	{attribute 'TcIecLibraryType'}
	{attribute 'external_name' := 'F_VN_AppendToContainer_ITcVnForwardIterator_GUID_EB72DC2C_3543_2E88_7126_C09EBB4E7DA0'}
	(* Append a single element (represented by an iterator)to a container. *)
	FUNCTION F_VN_AppendToContainer_ITcVnForwardIterator : HRESULT
	VAR_INPUT
		ipElement	:	ITcVnForwardIterator;	(* Single element to append to ipContainer *)
		ipContainer	:	ITcVnContainer;	(* Container to which the element(s) will be appended *)
		hrPrev	:	HRESULT;	(* HRESULT indicating the result of previous operations (If SUCCEEDED(hrPrev) equals false, no operation is executed.) *)
	END_VAR

END_FUNCTION

// Functions/Basic Container Operations/F_VN_AppendToContainer/F_VN_AppendToContainer_DINT

	{attribute 'TcIecLibraryType'}
	{attribute 'external_name' := 'F_VN_AppendToContainer_DINT_GUID_466F0C35_D3B5_2E85_68F4_3D84EB5E34A6'}
	(* Append a single element of type DINT to a container. *)
	FUNCTION F_VN_AppendToContainer_DINT : HRESULT
	VAR_INPUT
		nElement	:	DINT;	(* Single element to append to ipContainer *)
		ipContainer	:	ITcVnContainer;	(* Container to which the element will be appended *)
		hrPrev	:	HRESULT;	(* HRESULT indicating the result of previous operations (If SUCCEEDED(hrPrev) equals false, no operation is executed.) *)
	END_VAR

END_FUNCTION

// Functions/Basic Container Operations/F_VN_AppendToContainer/F_VN_AppendToContainer_INT

	{attribute 'TcIecLibraryType'}
	{attribute 'external_name' := 'F_VN_AppendToContainer_INT_GUID_9C2E93C7_B738_2FE7_7542_11A5629F66B3'}
	(* Append a single element of type INT to a container. *)
	FUNCTION F_VN_AppendToContainer_INT : HRESULT
	VAR_INPUT
		nElement	:	INT;	(* Single element to append to ipContainer *)
		ipContainer	:	ITcVnContainer;	(* Container to which the element will be appended *)
		hrPrev	:	HRESULT;	(* HRESULT indicating the result of previous operations (If SUCCEEDED(hrPrev) equals false, no operation is executed.) *)
	END_VAR

END_FUNCTION

// Functions/Basic Container Operations/F_VN_AppendToContainer/F_VN_AppendToContainer_ITcVnImage

	{attribute 'TcIecLibraryType'}
	{attribute 'external_name' := 'F_VN_AppendToContainer_ITcVnImage_GUID_1AC60876_C1A2_28F8_44E5_B78D9DB74DCF'}
	(* Append a single element of type ITcVnImage to a container. *)
	FUNCTION F_VN_AppendToContainer_ITcVnImage : HRESULT
	VAR_INPUT
		ipElement	:	ITcVnImage;	(* Single element to append to ipContainer *)
		ipContainer	:	ITcVnContainer;	(* Container to which the element will be appended *)
		hrPrev	:	HRESULT;	(* HRESULT indicating the result of previous operations (If SUCCEEDED(hrPrev) equals false, no operation is executed.) *)
	END_VAR

END_FUNCTION

// Functions/Basic Container Operations/F_VN_AppendToContainer/F_VN_AppendToContainer_LREAL

	{attribute 'TcIecLibraryType'}
	{attribute 'external_name' := 'F_VN_AppendToContainer_LREAL_GUID_B1A2121D_70A8_225D_5D75_B8BDFBCF299C'}
	(* Append a single element of type LREAL to a container. *)
	FUNCTION F_VN_AppendToContainer_LREAL : HRESULT
	VAR_INPUT
		fElement	:	LREAL;	(* Single element to append to ipContainer *)
		ipContainer	:	ITcVnContainer;	(* Container to which the element will be appended *)
		hrPrev	:	HRESULT;	(* HRESULT indicating the result of previous operations (If SUCCEEDED(hrPrev) equals false, no operation is executed.) *)
	END_VAR

END_FUNCTION

// Functions/Basic Container Operations/F_VN_AppendToContainer/F_VN_AppendToContainer_REAL

	{attribute 'TcIecLibraryType'}
	{attribute 'external_name' := 'F_VN_AppendToContainer_REAL_GUID_A8A7CA42_3B6F_24A9_44F1_7D2D9881B636'}
	(* Append a single element of type REAL to a container. *)
	FUNCTION F_VN_AppendToContainer_REAL : HRESULT
	VAR_INPUT
		fElement	:	REAL;	(* Single element to append to ipContainer *)
		ipContainer	:	ITcVnContainer;	(* Container to which the element will be appended *)
		hrPrev	:	HRESULT;	(* HRESULT indicating the result of previous operations (If SUCCEEDED(hrPrev) equals false, no operation is executed.) *)
	END_VAR

END_FUNCTION

// Functions/Basic Container Operations/F_VN_AppendToContainer/F_VN_AppendToContainer_SINT

	{attribute 'TcIecLibraryType'}
	{attribute 'external_name' := 'F_VN_AppendToContainer_SINT_GUID_2E825B48_89E4_2803_4016_10F4263A0344'}
	(* Append a single element of type SINT to a container. *)
	FUNCTION F_VN_AppendToContainer_SINT : HRESULT
	VAR_INPUT
		nElement	:	SINT;	(* Single element to append to ipContainer *)
		ipContainer	:	ITcVnContainer;	(* Container to which the element will be appended *)
		hrPrev	:	HRESULT;	(* HRESULT indicating the result of previous operations (If SUCCEEDED(hrPrev) equals false, no operation is executed.) *)
	END_VAR

END_FUNCTION

// Functions/Basic Container Operations/F_VN_AppendToContainer/F_VN_AppendToContainer_TcVnDMatch

	{attribute 'TcIecLibraryType'}
	{attribute 'external_name' := 'F_VN_AppendToContainer_TcVnDMatch_GUID_34846F37_CDB3_2F8C_4D45_929C7A1F5BBA'}
	(* Append a single element of type TcVnDMatch to a container. *)
	FUNCTION F_VN_AppendToContainer_TcVnDMatch : HRESULT
	VAR_IN_OUT
		stElement	:	TcVnDMatch;	(* Single element to append to ipContainer *)
	END_VAR
	VAR_INPUT
		ipContainer	:	ITcVnContainer;	(* Container to which the element will be appended *)
		hrPrev	:	HRESULT;	(* HRESULT indicating the result of previous operations (If SUCCEEDED(hrPrev) equals false, no operation is executed.) *)
	END_VAR

END_FUNCTION

// Functions/Basic Container Operations/F_VN_AppendToContainer/F_VN_AppendToContainer_TcVnKeyPoint

	{attribute 'TcIecLibraryType'}
	{attribute 'external_name' := 'F_VN_AppendToContainer_TcVnKeyPoint_GUID_DD1C6CD3_E38E_2AAF_58D6_28DA1BA2EF56'}
	(* Append a single element of type TcVnKeyPoint to a container. *)
	FUNCTION F_VN_AppendToContainer_TcVnKeyPoint : HRESULT
	VAR_IN_OUT
		stElement	:	TcVnKeyPoint;	(* Single element to append to ipContainer *)
	END_VAR
	VAR_INPUT
		ipContainer	:	ITcVnContainer;	(* Container to which the element will be appended *)
		hrPrev	:	HRESULT;	(* HRESULT indicating the result of previous operations (If SUCCEEDED(hrPrev) equals false, no operation is executed.) *)
	END_VAR

END_FUNCTION

// Functions/Basic Container Operations/F_VN_AppendToContainer/F_VN_AppendToContainer_TcVnPoint2_DINT

	{attribute 'TcIecLibraryType'}
	{attribute 'external_name' := 'F_VN_AppendToContainer_TcVnPoint2_DINT_GUID_E236D64B_774D_2339_6A19_DDD33484245C'}
	(* Append a single element of type TcVnPoint2_DINT to a container. *)
	FUNCTION F_VN_AppendToContainer_TcVnPoint2_DINT : HRESULT
	VAR_IN_OUT
		aElement	:	TcVnPoint2_DINT;	(* Single element to append to ipContainer *)
	END_VAR
	VAR_INPUT
		ipContainer	:	ITcVnContainer;	(* Container to which the element will be appended *)
		hrPrev	:	HRESULT;	(* HRESULT indicating the result of previous operations (If SUCCEEDED(hrPrev) equals false, no operation is executed.) *)
	END_VAR

END_FUNCTION

// Functions/Basic Container Operations/F_VN_AppendToContainer/F_VN_AppendToContainer_TcVnPoint2_LREAL

	{attribute 'TcIecLibraryType'}
	{attribute 'external_name' := 'F_VN_AppendToContainer_TcVnPoint2_LREAL_GUID_16F4346D_0CE3_2AEF_7282_0B6841F00F97'}
	(* Append a single element of type TcVnPoint2_LREAL to a container. *)
	FUNCTION F_VN_AppendToContainer_TcVnPoint2_LREAL : HRESULT
	VAR_IN_OUT
		aElement	:	TcVnPoint2_LREAL;	(* Single element to append to ipContainer *)
	END_VAR
	VAR_INPUT
		ipContainer	:	ITcVnContainer;	(* Container to which the element will be appended *)
		hrPrev	:	HRESULT;	(* HRESULT indicating the result of previous operations (If SUCCEEDED(hrPrev) equals false, no operation is executed.) *)
	END_VAR

END_FUNCTION

// Functions/Basic Container Operations/F_VN_AppendToContainer/F_VN_AppendToContainer_TcVnPoint2_REAL

	{attribute 'TcIecLibraryType'}
	{attribute 'external_name' := 'F_VN_AppendToContainer_TcVnPoint2_REAL_GUID_AF2054CF_707A_2EA1_59F4_ADBC6DC30FDD'}
	(* Append a single element of type TcVnPoint2_REAL to a container. *)
	FUNCTION F_VN_AppendToContainer_TcVnPoint2_REAL : HRESULT
	VAR_IN_OUT
		aElement	:	TcVnPoint2_REAL;	(* Single element to append to ipContainer *)
	END_VAR
	VAR_INPUT
		ipContainer	:	ITcVnContainer;	(* Container to which the element will be appended *)
		hrPrev	:	HRESULT;	(* HRESULT indicating the result of previous operations (If SUCCEEDED(hrPrev) equals false, no operation is executed.) *)
	END_VAR

END_FUNCTION

// Functions/Basic Container Operations/F_VN_AppendToContainer/F_VN_AppendToContainer_TcVnPoint3_LREAL

	{attribute 'TcIecLibraryType'}
	{attribute 'external_name' := 'F_VN_AppendToContainer_TcVnPoint3_LREAL_GUID_438155D5_801B_2D9E_780C_A41E6EF0A6F3'}
	(* Append a single element of type TcVnPoint3_LREAL to a container. *)
	FUNCTION F_VN_AppendToContainer_TcVnPoint3_LREAL : HRESULT
	VAR_IN_OUT
		aElement	:	TcVnPoint3_LREAL;	(* Single element to append to ipContainer *)
	END_VAR
	VAR_INPUT
		ipContainer	:	ITcVnContainer;	(* Container to which the element will be appended *)
		hrPrev	:	HRESULT;	(* HRESULT indicating the result of previous operations (If SUCCEEDED(hrPrev) equals false, no operation is executed.) *)
	END_VAR

END_FUNCTION

// Functions/Basic Container Operations/F_VN_AppendToContainer/F_VN_AppendToContainer_TcVnPoint3_REAL

	{attribute 'TcIecLibraryType'}
	{attribute 'external_name' := 'F_VN_AppendToContainer_TcVnPoint3_REAL_GUID_5F59C7E1_C02A_2A20_64DC_E35F15AD25C4'}
	(* Append a single element of type TcVnPoint3_REAL to a container. *)
	FUNCTION F_VN_AppendToContainer_TcVnPoint3_REAL : HRESULT
	VAR_IN_OUT
		aElement	:	TcVnPoint3_REAL;	(* Single element to append to ipContainer *)
	END_VAR
	VAR_INPUT
		ipContainer	:	ITcVnContainer;	(* Container to which the element will be appended *)
		hrPrev	:	HRESULT;	(* HRESULT indicating the result of previous operations (If SUCCEEDED(hrPrev) equals false, no operation is executed.) *)
	END_VAR

END_FUNCTION

// Functions/Basic Container Operations/F_VN_AppendToContainer/F_VN_AppendToContainer_TcVnRectangle_DINT

	{attribute 'TcIecLibraryType'}
	{attribute 'external_name' := 'F_VN_AppendToContainer_TcVnRectangle_DINT_GUID_4724E00F_EFEC_2862_725C_FE413D565967'}
	(* Append a single element of type TcVnRectangle_DINT to a container. *)
	FUNCTION F_VN_AppendToContainer_TcVnRectangle_DINT : HRESULT
	VAR_IN_OUT
		stElement	:	TcVnRectangle_DINT;	(* Single element to append to ipContainer *)
	END_VAR
	VAR_INPUT
		ipContainer	:	ITcVnContainer;	(* Container to which the element will be appended *)
		hrPrev	:	HRESULT;	(* HRESULT indicating the result of previous operations (If SUCCEEDED(hrPrev) equals false, no operation is executed.) *)
	END_VAR

END_FUNCTION

// Functions/Basic Container Operations/F_VN_AppendToContainer/F_VN_AppendToContainer_TcVnRotatedRectangle

	{attribute 'TcIecLibraryType'}
	{attribute 'external_name' := 'F_VN_AppendToContainer_TcVnRotatedRectangle_GUID_77E71F6F_47E9_24DA_6165_E73A8EF4D10B'}
	(* Append a single element of type TcVnRotatedRectangle to a container. *)
	FUNCTION F_VN_AppendToContainer_TcVnRotatedRectangle : HRESULT
	VAR_IN_OUT
		stElement	:	TcVnRotatedRectangle;	(* Single element to append to ipContainer *)
	END_VAR
	VAR_INPUT
		ipContainer	:	ITcVnContainer;	(* Container to which the element will be appended *)
		hrPrev	:	HRESULT;	(* HRESULT indicating the result of previous operations (If SUCCEEDED(hrPrev) equals false, no operation is executed.) *)
	END_VAR

END_FUNCTION

// Functions/Basic Container Operations/F_VN_AppendToContainer/F_VN_AppendToContainer_TcVnVector2_DINT

	{attribute 'TcIecLibraryType'}
	{attribute 'external_name' := 'F_VN_AppendToContainer_TcVnVector2_DINT_GUID_C23FB6C1_69D6_29E0_479F_7FD94985AF4C'}
	(* Append a single element of type TcVnVector2_DINT to a container. *)
	FUNCTION F_VN_AppendToContainer_TcVnVector2_DINT : HRESULT
	VAR_IN_OUT
		aElement	:	TcVnVector2_DINT;	(* Single element to append to ipContainer *)
	END_VAR
	VAR_INPUT
		ipContainer	:	ITcVnContainer;	(* Container to which the element will be appended *)
		hrPrev	:	HRESULT;	(* HRESULT indicating the result of previous operations (If SUCCEEDED(hrPrev) equals false, no operation is executed.) *)
	END_VAR

END_FUNCTION

// Functions/Basic Container Operations/F_VN_AppendToContainer/F_VN_AppendToContainer_TcVnVector2_INT

	{attribute 'TcIecLibraryType'}
	{attribute 'external_name' := 'F_VN_AppendToContainer_TcVnVector2_INT_GUID_8095F8C5_D9A4_2714_5F67_D5F454AA922A'}
	(* Append a single element of type TcVnVector2_INT to a container. *)
	FUNCTION F_VN_AppendToContainer_TcVnVector2_INT : HRESULT
	VAR_IN_OUT
		aElement	:	TcVnVector2_INT;	(* Single element to append to ipContainer *)
	END_VAR
	VAR_INPUT
		ipContainer	:	ITcVnContainer;	(* Container to which the element will be appended *)
		hrPrev	:	HRESULT;	(* HRESULT indicating the result of previous operations (If SUCCEEDED(hrPrev) equals false, no operation is executed.) *)
	END_VAR

END_FUNCTION

// Functions/Basic Container Operations/F_VN_AppendToContainer/F_VN_AppendToContainer_TcVnVector2_REAL

	{attribute 'TcIecLibraryType'}
	{attribute 'external_name' := 'F_VN_AppendToContainer_TcVnVector2_REAL_GUID_4925EF9F_1A70_2872_599C_619CA5976C40'}
	(* Append a single element of type TcVnVector2_REAL to a container. *)
	FUNCTION F_VN_AppendToContainer_TcVnVector2_REAL : HRESULT
	VAR_IN_OUT
		aElement	:	TcVnVector2_REAL;	(* Single element to append to ipContainer *)
	END_VAR
	VAR_INPUT
		ipContainer	:	ITcVnContainer;	(* Container to which the element will be appended *)
		hrPrev	:	HRESULT;	(* HRESULT indicating the result of previous operations (If SUCCEEDED(hrPrev) equals false, no operation is executed.) *)
	END_VAR

END_FUNCTION

// Functions/Basic Container Operations/F_VN_AppendToContainer/F_VN_AppendToContainer_TcVnVector2_SINT

	{attribute 'TcIecLibraryType'}
	{attribute 'external_name' := 'F_VN_AppendToContainer_TcVnVector2_SINT_GUID_31CFB0CF_5D30_23E7_78F5_3FE68E6ABFCD'}
	(* Append a single element of type TcVnVector2_SINT to a container. *)
	FUNCTION F_VN_AppendToContainer_TcVnVector2_SINT : HRESULT
	VAR_IN_OUT
		aElement	:	TcVnVector2_SINT;	(* Single element to append to ipContainer *)
	END_VAR
	VAR_INPUT
		ipContainer	:	ITcVnContainer;	(* Container to which the element will be appended *)
		hrPrev	:	HRESULT;	(* HRESULT indicating the result of previous operations (If SUCCEEDED(hrPrev) equals false, no operation is executed.) *)
	END_VAR

END_FUNCTION

// Functions/Basic Container Operations/F_VN_AppendToContainer/F_VN_AppendToContainer_TcVnVector2_UINT

	{attribute 'TcIecLibraryType'}
	{attribute 'external_name' := 'F_VN_AppendToContainer_TcVnVector2_UINT_GUID_E6467BA2_FB3C_202A_4A01_9C9813DD37CA'}
	(* Append a single element of type TcVnVector2_UINT to a container. *)
	FUNCTION F_VN_AppendToContainer_TcVnVector2_UINT : HRESULT
	VAR_IN_OUT
		aElement	:	TcVnVector2_UINT;	(* Single element to append to ipContainer *)
	END_VAR
	VAR_INPUT
		ipContainer	:	ITcVnContainer;	(* Container to which the element will be appended *)
		hrPrev	:	HRESULT;	(* HRESULT indicating the result of previous operations (If SUCCEEDED(hrPrev) equals false, no operation is executed.) *)
	END_VAR

END_FUNCTION

// Functions/Basic Container Operations/F_VN_AppendToContainer/F_VN_AppendToContainer_TcVnVector2_USINT

	{attribute 'TcIecLibraryType'}
	{attribute 'external_name' := 'F_VN_AppendToContainer_TcVnVector2_USINT_GUID_4C52AFE9_65D3_2664_4952_BF781569C1D3'}
	(* Append a single element of type TcVnVector2_USINT to a container. *)
	FUNCTION F_VN_AppendToContainer_TcVnVector2_USINT : HRESULT
	VAR_IN_OUT
		aElement	:	TcVnVector2_USINT;	(* Single element to append to ipContainer *)
	END_VAR
	VAR_INPUT
		ipContainer	:	ITcVnContainer;	(* Container to which the element will be appended *)
		hrPrev	:	HRESULT;	(* HRESULT indicating the result of previous operations (If SUCCEEDED(hrPrev) equals false, no operation is executed.) *)
	END_VAR

END_FUNCTION

// Functions/Basic Container Operations/F_VN_AppendToContainer/F_VN_AppendToContainer_TcVnVector3_INT

	{attribute 'TcIecLibraryType'}
	{attribute 'external_name' := 'F_VN_AppendToContainer_TcVnVector3_INT_GUID_05D2B112_0D58_2E07_4C5E_A3CD17160E9A'}
	(* Append a single element of type TcVnVector3_INT to a container. *)
	FUNCTION F_VN_AppendToContainer_TcVnVector3_INT : HRESULT
	VAR_IN_OUT
		aElement	:	TcVnVector3_INT;	(* Single element to append to ipContainer *)
	END_VAR
	VAR_INPUT
		ipContainer	:	ITcVnContainer;	(* Container to which the element will be appended *)
		hrPrev	:	HRESULT;	(* HRESULT indicating the result of previous operations (If SUCCEEDED(hrPrev) equals false, no operation is executed.) *)
	END_VAR

END_FUNCTION

// Functions/Basic Container Operations/F_VN_AppendToContainer/F_VN_AppendToContainer_TcVnVector3_REAL

	{attribute 'TcIecLibraryType'}
	{attribute 'external_name' := 'F_VN_AppendToContainer_TcVnVector3_REAL_GUID_514006DF_962C_2E5C_69E4_43541FF1F6C6'}
	(* Append a single element of type TcVnVector3_REAL to a container. *)
	FUNCTION F_VN_AppendToContainer_TcVnVector3_REAL : HRESULT
	VAR_IN_OUT
		aElement	:	TcVnVector3_REAL;	(* Single element to append to ipContainer *)
	END_VAR
	VAR_INPUT
		ipContainer	:	ITcVnContainer;	(* Container to which the element will be appended *)
		hrPrev	:	HRESULT;	(* HRESULT indicating the result of previous operations (If SUCCEEDED(hrPrev) equals false, no operation is executed.) *)
	END_VAR

END_FUNCTION

// Functions/Basic Container Operations/F_VN_AppendToContainer/F_VN_AppendToContainer_TcVnVector3_SINT

	{attribute 'TcIecLibraryType'}
	{attribute 'external_name' := 'F_VN_AppendToContainer_TcVnVector3_SINT_GUID_4338E815_E137_2C69_40A4_187C43F3E877'}
	(* Append a single element of type TcVnVector3_SINT to a container. *)
	FUNCTION F_VN_AppendToContainer_TcVnVector3_SINT : HRESULT
	VAR_IN_OUT
		aElement	:	TcVnVector3_SINT;	(* Single element to append to ipContainer *)
	END_VAR
	VAR_INPUT
		ipContainer	:	ITcVnContainer;	(* Container to which the element will be appended *)
		hrPrev	:	HRESULT;	(* HRESULT indicating the result of previous operations (If SUCCEEDED(hrPrev) equals false, no operation is executed.) *)
	END_VAR

END_FUNCTION

// Functions/Basic Container Operations/F_VN_AppendToContainer/F_VN_AppendToContainer_TcVnVector3_UINT

	{attribute 'TcIecLibraryType'}
	{attribute 'external_name' := 'F_VN_AppendToContainer_TcVnVector3_UINT_GUID_758EB63E_2A0A_2104_750E_5DD44351B258'}
	(* Append a single element of type TcVnVector3_UINT to a container. *)
	FUNCTION F_VN_AppendToContainer_TcVnVector3_UINT : HRESULT
	VAR_IN_OUT
		aElement	:	TcVnVector3_UINT;	(* Single element to append to ipContainer *)
	END_VAR
	VAR_INPUT
		ipContainer	:	ITcVnContainer;	(* Container to which the element will be appended *)
		hrPrev	:	HRESULT;	(* HRESULT indicating the result of previous operations (If SUCCEEDED(hrPrev) equals false, no operation is executed.) *)
	END_VAR

END_FUNCTION

// Functions/Basic Container Operations/F_VN_AppendToContainer/F_VN_AppendToContainer_TcVnVector3_USINT

	{attribute 'TcIecLibraryType'}
	{attribute 'external_name' := 'F_VN_AppendToContainer_TcVnVector3_USINT_GUID_08EE0EEE_C71B_2ED9_5959_1E12B89BC7B4'}
	(* Append a single element of type TcVnVector3_USINT to a container. *)
	FUNCTION F_VN_AppendToContainer_TcVnVector3_USINT : HRESULT
	VAR_IN_OUT
		aElement	:	TcVnVector3_USINT;	(* Single element to append to ipContainer *)
	END_VAR
	VAR_INPUT
		ipContainer	:	ITcVnContainer;	(* Container to which the element will be appended *)
		hrPrev	:	HRESULT;	(* HRESULT indicating the result of previous operations (If SUCCEEDED(hrPrev) equals false, no operation is executed.) *)
	END_VAR

END_FUNCTION

// Functions/Basic Container Operations/F_VN_AppendToContainer/F_VN_AppendToContainer_TcVnVector4_DINT

	{attribute 'TcIecLibraryType'}
	{attribute 'external_name' := 'F_VN_AppendToContainer_TcVnVector4_DINT_GUID_083F1B4F_E0BF_20EA_4234_CF3DA9D51929'}
	(* Append a single element of type TcVnVector4_DINT to a container. *)
	FUNCTION F_VN_AppendToContainer_TcVnVector4_DINT : HRESULT
	VAR_IN_OUT
		aElement	:	TcVnVector4_DINT;	(* Single element to append to ipContainer *)
	END_VAR
	VAR_INPUT
		ipContainer	:	ITcVnContainer;	(* Container to which the element will be appended *)
		hrPrev	:	HRESULT;	(* HRESULT indicating the result of previous operations (If SUCCEEDED(hrPrev) equals false, no operation is executed.) *)
	END_VAR

END_FUNCTION

// Functions/Basic Container Operations/F_VN_AppendToContainer/F_VN_AppendToContainer_TcVnVector4_INT

	{attribute 'TcIecLibraryType'}
	{attribute 'external_name' := 'F_VN_AppendToContainer_TcVnVector4_INT_GUID_0322E615_B58F_2529_4092_135330AE55A7'}
	(* Append a single element of type TcVnVector4_INT to a container. *)
	FUNCTION F_VN_AppendToContainer_TcVnVector4_INT : HRESULT
	VAR_IN_OUT
		aElement	:	TcVnVector4_INT;	(* Single element to append to ipContainer *)
	END_VAR
	VAR_INPUT
		ipContainer	:	ITcVnContainer;	(* Container to which the element will be appended *)
		hrPrev	:	HRESULT;	(* HRESULT indicating the result of previous operations (If SUCCEEDED(hrPrev) equals false, no operation is executed.) *)
	END_VAR

END_FUNCTION

// Functions/Basic Container Operations/F_VN_AppendToContainer/F_VN_AppendToContainer_TcVnVector4_LREAL

	{attribute 'TcIecLibraryType'}
	{attribute 'external_name' := 'F_VN_AppendToContainer_TcVnVector4_LREAL_GUID_681DC552_1562_26E2_4E2A_2A3742704EEB'}
	(* Append a single element of type TcVnVector4_LREAL to a container. *)
	FUNCTION F_VN_AppendToContainer_TcVnVector4_LREAL : HRESULT
	VAR_IN_OUT
		aElement	:	TcVnVector4_LREAL;	(* Single element to append to ipContainer *)
	END_VAR
	VAR_INPUT
		ipContainer	:	ITcVnContainer;	(* Container to which the element will be appended *)
		hrPrev	:	HRESULT;	(* HRESULT indicating the result of previous operations (If SUCCEEDED(hrPrev) equals false, no operation is executed.) *)
	END_VAR

END_FUNCTION

// Functions/Basic Container Operations/F_VN_AppendToContainer/F_VN_AppendToContainer_TcVnVector4_REAL

	{attribute 'TcIecLibraryType'}
	{attribute 'external_name' := 'F_VN_AppendToContainer_TcVnVector4_REAL_GUID_C3C2BE2E_4B29_2FE9_5F64_0CA6798DF02D'}
	(* Append a single element of type TcVnVector4_REAL to a container. *)
	FUNCTION F_VN_AppendToContainer_TcVnVector4_REAL : HRESULT
	VAR_IN_OUT
		aElement	:	TcVnVector4_REAL;	(* Single element to append to ipContainer *)
	END_VAR
	VAR_INPUT
		ipContainer	:	ITcVnContainer;	(* Container to which the element will be appended *)
		hrPrev	:	HRESULT;	(* HRESULT indicating the result of previous operations (If SUCCEEDED(hrPrev) equals false, no operation is executed.) *)
	END_VAR

END_FUNCTION

// Functions/Basic Container Operations/F_VN_AppendToContainer/F_VN_AppendToContainer_TcVnVector4_SINT

	{attribute 'TcIecLibraryType'}
	{attribute 'external_name' := 'F_VN_AppendToContainer_TcVnVector4_SINT_GUID_8FC9D3FA_1CE7_2907_4A68_5B1791743FF4'}
	(* Append a single element of type TcVnVector4_SINT to a container. *)
	FUNCTION F_VN_AppendToContainer_TcVnVector4_SINT : HRESULT
	VAR_IN_OUT
		aElement	:	TcVnVector4_SINT;	(* Single element to append to ipContainer *)
	END_VAR
	VAR_INPUT
		ipContainer	:	ITcVnContainer;	(* Container to which the element will be appended *)
		hrPrev	:	HRESULT;	(* HRESULT indicating the result of previous operations (If SUCCEEDED(hrPrev) equals false, no operation is executed.) *)
	END_VAR

END_FUNCTION

// Functions/Basic Container Operations/F_VN_AppendToContainer/F_VN_AppendToContainer_TcVnVector4_UINT

	{attribute 'TcIecLibraryType'}
	{attribute 'external_name' := 'F_VN_AppendToContainer_TcVnVector4_UINT_GUID_83BE3591_1DA5_2EF5_7310_4ED88571AA65'}
	(* Append a single element of type TcVnVector4_UINT to a container. *)
	FUNCTION F_VN_AppendToContainer_TcVnVector4_UINT : HRESULT
	VAR_IN_OUT
		aElement	:	TcVnVector4_UINT;	(* Single element to append to ipContainer *)
	END_VAR
	VAR_INPUT
		ipContainer	:	ITcVnContainer;	(* Container to which the element will be appended *)
		hrPrev	:	HRESULT;	(* HRESULT indicating the result of previous operations (If SUCCEEDED(hrPrev) equals false, no operation is executed.) *)
	END_VAR

END_FUNCTION

// Functions/Basic Container Operations/F_VN_AppendToContainer/F_VN_AppendToContainer_TcVnVector4_USINT

	{attribute 'TcIecLibraryType'}
	{attribute 'external_name' := 'F_VN_AppendToContainer_TcVnVector4_USINT_GUID_6F87F9FC_F9CB_23B6_6496_A174F0A1309B'}
	(* Append a single element of type TcVnVector4_USINT to a container. *)
	FUNCTION F_VN_AppendToContainer_TcVnVector4_USINT : HRESULT
	VAR_IN_OUT
		aElement	:	TcVnVector4_USINT;	(* Single element to append to ipContainer *)
	END_VAR
	VAR_INPUT
		ipContainer	:	ITcVnContainer;	(* Container to which the element will be appended *)
		hrPrev	:	HRESULT;	(* HRESULT indicating the result of previous operations (If SUCCEEDED(hrPrev) equals false, no operation is executed.) *)
	END_VAR

END_FUNCTION

// Functions/Basic Container Operations/F_VN_AppendToContainer/F_VN_AppendToContainer_UDINT

	{attribute 'TcIecLibraryType'}
	{attribute 'external_name' := 'F_VN_AppendToContainer_UDINT_GUID_8470ED3B_0039_2C3C_7E1C_C11327C98C97'}
	(* Append a single element of type UDINT to a container. *)
	FUNCTION F_VN_AppendToContainer_UDINT : HRESULT
	VAR_INPUT
		nElement	:	UDINT;	(* Single element to append to ipContainer *)
		ipContainer	:	ITcVnContainer;	(* Container to which the element will be appended *)
		hrPrev	:	HRESULT;	(* HRESULT indicating the result of previous operations (If SUCCEEDED(hrPrev) equals false, no operation is executed.) *)
	END_VAR

END_FUNCTION

// Functions/Basic Container Operations/F_VN_AppendToContainer/F_VN_AppendToContainer_UINT

	{attribute 'TcIecLibraryType'}
	{attribute 'external_name' := 'F_VN_AppendToContainer_UINT_GUID_3E3BAFD3_4B5E_2BD9_48BE_994F27FEBDF9'}
	(* Append a single element of type UINT to a container. *)
	FUNCTION F_VN_AppendToContainer_UINT : HRESULT
	VAR_INPUT
		nElement	:	UINT;	(* Single element to append to ipContainer *)
		ipContainer	:	ITcVnContainer;	(* Container to which the element will be appended *)
		hrPrev	:	HRESULT;	(* HRESULT indicating the result of previous operations (If SUCCEEDED(hrPrev) equals false, no operation is executed.) *)
	END_VAR

END_FUNCTION

// Functions/Basic Container Operations/F_VN_AppendToContainer/F_VN_AppendToContainer_ULINT

	{attribute 'TcIecLibraryType'}
	{attribute 'external_name' := 'F_VN_AppendToContainer_ULINT_GUID_B226B100_672F_2892_4B91_CCC667888FCA'}
	(* Append a single element of type ULINT to a container. *)
	FUNCTION F_VN_AppendToContainer_ULINT : HRESULT
	VAR_INPUT
		nElement	:	ULINT;	(* Single element to append to ipContainer *)
		ipContainer	:	ITcVnContainer;	(* Container to which the element will be appended *)
		hrPrev	:	HRESULT;	(* HRESULT indicating the result of previous operations (If SUCCEEDED(hrPrev) equals false, no operation is executed.) *)
	END_VAR

END_FUNCTION

// Functions/Basic Container Operations/F_VN_AppendToContainer/F_VN_AppendToContainer_USINT

	{attribute 'TcIecLibraryType'}
	{attribute 'external_name' := 'F_VN_AppendToContainer_USINT_GUID_0CA19091_82AA_2F8A_54F9_1345671338BF'}
	(* Append a single element of type USINT to a container. *)
	FUNCTION F_VN_AppendToContainer_USINT : HRESULT
	VAR_INPUT
		nElement	:	USINT;	(* Single element to append to ipContainer *)
		ipContainer	:	ITcVnContainer;	(* Container to which the element will be appended *)
		hrPrev	:	HRESULT;	(* HRESULT indicating the result of previous operations (If SUCCEEDED(hrPrev) equals false, no operation is executed.) *)
	END_VAR

END_FUNCTION

// Functions/Basic Container Operations/F_VN_FillContainer/F_VN_FillContainer_DINT

	{attribute 'TcIecLibraryType'}
	{attribute 'external_name' := 'F_VN_FillContainer_DINT_GUID_083E9E6C_5222_2ABE_5F48_D869D6266B91'}
	(* Fill the container with the specified value. Only possible for containers with basic elements. *)
	FUNCTION F_VN_FillContainer_DINT : HRESULT
	VAR_INPUT
		ipContainer	:	ITcVnContainer;	(* Container with basic elements *)
		nValue	:	DINT;	(* Value to set the container elements *)
		hrPrev	:	HRESULT;	(* HRESULT indicating the result of previous operations (If SUCCEEDED(hrPrev) equals false, no operation is executed.) *)
	END_VAR

END_FUNCTION

// Functions/Basic Container Operations/F_VN_FillContainer/F_VN_FillContainer_INT

	{attribute 'TcIecLibraryType'}
	{attribute 'external_name' := 'F_VN_FillContainer_INT_GUID_8ED3136D_AC68_2FDD_4634_FD980A7E826E'}
	(* Fill the container with the specified value. Only possible for containers with basic elements. *)
	FUNCTION F_VN_FillContainer_INT : HRESULT
	VAR_INPUT
		ipContainer	:	ITcVnContainer;	(* Container with basic elements *)
		nValue	:	INT;	(* Value to set the container elements *)
		hrPrev	:	HRESULT;	(* HRESULT indicating the result of previous operations (If SUCCEEDED(hrPrev) equals false, no operation is executed.) *)
	END_VAR

END_FUNCTION

// Functions/Basic Container Operations/F_VN_FillContainer/F_VN_FillContainer_ITcVnImage

	{attribute 'TcIecLibraryType'}
	{attribute 'external_name' := 'F_VN_FillContainer_ITcVnImage_GUID_22A97681_F470_26EA_685A_388B886A33A4'}
	(* Fill the container with the specified value. Only possible for containers with basic elements. *)
	FUNCTION F_VN_FillContainer_ITcVnImage : HRESULT
	VAR_INPUT
		ipContainer	:	ITcVnContainer;	(* Container with basic elements *)
		ipValue	:	ITcVnImage;	(* Value to set the container elements *)
		hrPrev	:	HRESULT;	(* HRESULT indicating the result of previous operations (If SUCCEEDED(hrPrev) equals false, no operation is executed.) *)
	END_VAR

END_FUNCTION

// Functions/Basic Container Operations/F_VN_FillContainer/F_VN_FillContainer_LREAL

	{attribute 'TcIecLibraryType'}
	{attribute 'external_name' := 'F_VN_FillContainer_LREAL_GUID_8D3F02AD_A4BF_2560_5EEB_A5E316D08C86'}
	(* Fill the container with the specified value. Only possible for containers with basic elements. *)
	FUNCTION F_VN_FillContainer_LREAL : HRESULT
	VAR_INPUT
		ipContainer	:	ITcVnContainer;	(* Container with basic elements *)
		fValue	:	LREAL;	(* Value to set the container elements *)
		hrPrev	:	HRESULT;	(* HRESULT indicating the result of previous operations (If SUCCEEDED(hrPrev) equals false, no operation is executed.) *)
	END_VAR

END_FUNCTION

// Functions/Basic Container Operations/F_VN_FillContainer/F_VN_FillContainer_REAL

	{attribute 'TcIecLibraryType'}
	{attribute 'external_name' := 'F_VN_FillContainer_REAL_GUID_D0352CFF_BD98_2FB9_6053_3682B51A45BC'}
	(* Fill the container with the specified value. Only possible for containers with basic elements. *)
	FUNCTION F_VN_FillContainer_REAL : HRESULT
	VAR_INPUT
		ipContainer	:	ITcVnContainer;	(* Container with basic elements *)
		fValue	:	REAL;	(* Value to set the container elements *)
		hrPrev	:	HRESULT;	(* HRESULT indicating the result of previous operations (If SUCCEEDED(hrPrev) equals false, no operation is executed.) *)
	END_VAR

END_FUNCTION

// Functions/Basic Container Operations/F_VN_FillContainer/F_VN_FillContainer_SINT

	{attribute 'TcIecLibraryType'}
	{attribute 'external_name' := 'F_VN_FillContainer_SINT_GUID_F7096BE8_CA7B_2D9D_52DC_053DD750BF89'}
	(* Fill the container with the specified value. Only possible for containers with basic elements. *)
	FUNCTION F_VN_FillContainer_SINT : HRESULT
	VAR_INPUT
		ipContainer	:	ITcVnContainer;	(* Container with basic elements *)
		nValue	:	SINT;	(* Value to set the container elements *)
		hrPrev	:	HRESULT;	(* HRESULT indicating the result of previous operations (If SUCCEEDED(hrPrev) equals false, no operation is executed.) *)
	END_VAR

END_FUNCTION

// Functions/Basic Container Operations/F_VN_FillContainer/F_VN_FillContainer_TcVnDMatch

	{attribute 'TcIecLibraryType'}
	{attribute 'external_name' := 'F_VN_FillContainer_TcVnDMatch_GUID_9AC9DFDA_B578_29CB_55F9_C4FCEA2CCD41'}
	(* Fill the container with the specified value. Only possible for containers with basic elements. *)
	FUNCTION F_VN_FillContainer_TcVnDMatch : HRESULT
	VAR_INPUT
		ipContainer	:	ITcVnContainer;	(* Container with basic elements *)
	END_VAR
	VAR_IN_OUT
		stValue	:	TcVnDMatch;	(* Value to set the container elements *)
	END_VAR
	VAR_INPUT
		hrPrev	:	HRESULT;	(* HRESULT indicating the result of previous operations (If SUCCEEDED(hrPrev) equals false, no operation is executed.) *)
	END_VAR

END_FUNCTION

// Functions/Basic Container Operations/F_VN_FillContainer/F_VN_FillContainer_TcVnKeyPoint

	{attribute 'TcIecLibraryType'}
	{attribute 'external_name' := 'F_VN_FillContainer_TcVnKeyPoint_GUID_107991CE_CBF7_2C98_5C18_AF43F9BA9556'}
	(* Fill the container with the specified value. Only possible for containers with basic elements. *)
	FUNCTION F_VN_FillContainer_TcVnKeyPoint : HRESULT
	VAR_INPUT
		ipContainer	:	ITcVnContainer;	(* Container with basic elements *)
	END_VAR
	VAR_IN_OUT
		stValue	:	TcVnKeyPoint;	(* Value to set the container elements *)
	END_VAR
	VAR_INPUT
		hrPrev	:	HRESULT;	(* HRESULT indicating the result of previous operations (If SUCCEEDED(hrPrev) equals false, no operation is executed.) *)
	END_VAR

END_FUNCTION

// Functions/Basic Container Operations/F_VN_FillContainer/F_VN_FillContainer_TcVnPoint2_DINT

	{attribute 'TcIecLibraryType'}
	{attribute 'external_name' := 'F_VN_FillContainer_TcVnPoint2_DINT_GUID_0AE65E92_37EC_24E8_53D5_0D613C34FAB7'}
	(* Fill the container with the specified value. Only possible for containers with basic elements. *)
	FUNCTION F_VN_FillContainer_TcVnPoint2_DINT : HRESULT
	VAR_INPUT
		ipContainer	:	ITcVnContainer;	(* Container with basic elements *)
	END_VAR
	VAR_IN_OUT
		aValue	:	TcVnPoint2_DINT;	(* Value to set the container elements *)
	END_VAR
	VAR_INPUT
		hrPrev	:	HRESULT;	(* HRESULT indicating the result of previous operations (If SUCCEEDED(hrPrev) equals false, no operation is executed.) *)
	END_VAR

END_FUNCTION

// Functions/Basic Container Operations/F_VN_FillContainer/F_VN_FillContainer_TcVnPoint2_LREAL

	{attribute 'TcIecLibraryType'}
	{attribute 'external_name' := 'F_VN_FillContainer_TcVnPoint2_LREAL_GUID_AA3BABFF_E9F8_2284_7A63_D6343B715275'}
	(* Fill the container with the specified value. Only possible for containers with basic elements. *)
	FUNCTION F_VN_FillContainer_TcVnPoint2_LREAL : HRESULT
	VAR_INPUT
		ipContainer	:	ITcVnContainer;	(* Container with basic elements *)
	END_VAR
	VAR_IN_OUT
		aValue	:	TcVnPoint2_LREAL;	(* Value to set the container elements *)
	END_VAR
	VAR_INPUT
		hrPrev	:	HRESULT;	(* HRESULT indicating the result of previous operations (If SUCCEEDED(hrPrev) equals false, no operation is executed.) *)
	END_VAR

END_FUNCTION

// Functions/Basic Container Operations/F_VN_FillContainer/F_VN_FillContainer_TcVnPoint2_REAL

	{attribute 'TcIecLibraryType'}
	{attribute 'external_name' := 'F_VN_FillContainer_TcVnPoint2_REAL_GUID_058A1755_37CF_2846_5587_BDB7740DB546'}
	(* Fill the container with the specified value. Only possible for containers with basic elements. *)
	FUNCTION F_VN_FillContainer_TcVnPoint2_REAL : HRESULT
	VAR_INPUT
		ipContainer	:	ITcVnContainer;	(* Container with basic elements *)
	END_VAR
	VAR_IN_OUT
		aValue	:	TcVnPoint2_REAL;	(* Value to set the container elements *)
	END_VAR
	VAR_INPUT
		hrPrev	:	HRESULT;	(* HRESULT indicating the result of previous operations (If SUCCEEDED(hrPrev) equals false, no operation is executed.) *)
	END_VAR

END_FUNCTION

// Functions/Basic Container Operations/F_VN_FillContainer/F_VN_FillContainer_TcVnPoint3_LREAL

	{attribute 'TcIecLibraryType'}
	{attribute 'external_name' := 'F_VN_FillContainer_TcVnPoint3_LREAL_GUID_FECA52C2_308A_2C33_6354_98D6D1E872F0'}
	(* Fill the container with the specified value. Only possible for containers with basic elements. *)
	FUNCTION F_VN_FillContainer_TcVnPoint3_LREAL : HRESULT
	VAR_INPUT
		ipContainer	:	ITcVnContainer;	(* Container with basic elements *)
	END_VAR
	VAR_IN_OUT
		aValue	:	TcVnPoint3_LREAL;	(* Value to set the container elements *)
	END_VAR
	VAR_INPUT
		hrPrev	:	HRESULT;	(* HRESULT indicating the result of previous operations (If SUCCEEDED(hrPrev) equals false, no operation is executed.) *)
	END_VAR

END_FUNCTION

// Functions/Basic Container Operations/F_VN_FillContainer/F_VN_FillContainer_TcVnPoint3_REAL

	{attribute 'TcIecLibraryType'}
	{attribute 'external_name' := 'F_VN_FillContainer_TcVnPoint3_REAL_GUID_1F43B1B1_5F35_2D89_59FA_81F0769BFFB3'}
	(* Fill the container with the specified value. Only possible for containers with basic elements. *)
	FUNCTION F_VN_FillContainer_TcVnPoint3_REAL : HRESULT
	VAR_INPUT
		ipContainer	:	ITcVnContainer;	(* Container with basic elements *)
	END_VAR
	VAR_IN_OUT
		aValue	:	TcVnPoint3_REAL;	(* Value to set the container elements *)
	END_VAR
	VAR_INPUT
		hrPrev	:	HRESULT;	(* HRESULT indicating the result of previous operations (If SUCCEEDED(hrPrev) equals false, no operation is executed.) *)
	END_VAR

END_FUNCTION

// Functions/Basic Container Operations/F_VN_FillContainer/F_VN_FillContainer_TcVnRectangle_DINT

	{attribute 'TcIecLibraryType'}
	{attribute 'external_name' := 'F_VN_FillContainer_TcVnRectangle_DINT_GUID_6F8A925D_1642_2178_7DE5_A6DFA466B955'}
	(* Fill the container with the specified value. Only possible for containers with basic elements. *)
	FUNCTION F_VN_FillContainer_TcVnRectangle_DINT : HRESULT
	VAR_INPUT
		ipContainer	:	ITcVnContainer;	(* Container with basic elements *)
	END_VAR
	VAR_IN_OUT
		stValue	:	TcVnRectangle_DINT;	(* Value to set the container elements *)
	END_VAR
	VAR_INPUT
		hrPrev	:	HRESULT;	(* HRESULT indicating the result of previous operations (If SUCCEEDED(hrPrev) equals false, no operation is executed.) *)
	END_VAR

END_FUNCTION

// Functions/Basic Container Operations/F_VN_FillContainer/F_VN_FillContainer_TcVnRotatedRectangle

	{attribute 'TcIecLibraryType'}
	{attribute 'external_name' := 'F_VN_FillContainer_TcVnRotatedRectangle_GUID_3A39EDD0_173C_209A_7C32_6015F26F980F'}
	(* Fill the container with the specified value. Only possible for containers with basic elements. *)
	FUNCTION F_VN_FillContainer_TcVnRotatedRectangle : HRESULT
	VAR_INPUT
		ipContainer	:	ITcVnContainer;	(* Container with basic elements *)
	END_VAR
	VAR_IN_OUT
		stValue	:	TcVnRotatedRectangle;	(* Value to set the container elements *)
	END_VAR
	VAR_INPUT
		hrPrev	:	HRESULT;	(* HRESULT indicating the result of previous operations (If SUCCEEDED(hrPrev) equals false, no operation is executed.) *)
	END_VAR

END_FUNCTION

// Functions/Basic Container Operations/F_VN_FillContainer/F_VN_FillContainer_TcVnVector2_DINT

	{attribute 'TcIecLibraryType'}
	{attribute 'external_name' := 'F_VN_FillContainer_TcVnVector2_DINT_GUID_551E9BEE_BA99_2B02_7ADD_C292B12725EE'}
	(* Fill the container with the specified value. Only possible for containers with basic elements. *)
	FUNCTION F_VN_FillContainer_TcVnVector2_DINT : HRESULT
	VAR_INPUT
		ipContainer	:	ITcVnContainer;	(* Container with basic elements *)
	END_VAR
	VAR_IN_OUT
		aValue	:	TcVnVector2_DINT;	(* Value to set the container elements *)
	END_VAR
	VAR_INPUT
		hrPrev	:	HRESULT;	(* HRESULT indicating the result of previous operations (If SUCCEEDED(hrPrev) equals false, no operation is executed.) *)
	END_VAR

END_FUNCTION

// Functions/Basic Container Operations/F_VN_FillContainer/F_VN_FillContainer_TcVnVector2_INT

	{attribute 'TcIecLibraryType'}
	{attribute 'external_name' := 'F_VN_FillContainer_TcVnVector2_INT_GUID_85BEE863_02C8_26B6_4CCA_D223532C0910'}
	(* Fill the container with the specified value. Only possible for containers with basic elements. *)
	FUNCTION F_VN_FillContainer_TcVnVector2_INT : HRESULT
	VAR_INPUT
		ipContainer	:	ITcVnContainer;	(* Container with basic elements *)
	END_VAR
	VAR_IN_OUT
		aValue	:	TcVnVector2_INT;	(* Value to set the container elements *)
	END_VAR
	VAR_INPUT
		hrPrev	:	HRESULT;	(* HRESULT indicating the result of previous operations (If SUCCEEDED(hrPrev) equals false, no operation is executed.) *)
	END_VAR

END_FUNCTION

// Functions/Basic Container Operations/F_VN_FillContainer/F_VN_FillContainer_TcVnVector2_REAL

	{attribute 'TcIecLibraryType'}
	{attribute 'external_name' := 'F_VN_FillContainer_TcVnVector2_REAL_GUID_C2DFFCFC_A4D7_25BD_49D7_3DCABE4B2F8A'}
	(* Fill the container with the specified value. Only possible for containers with basic elements. *)
	FUNCTION F_VN_FillContainer_TcVnVector2_REAL : HRESULT
	VAR_INPUT
		ipContainer	:	ITcVnContainer;	(* Container with basic elements *)
	END_VAR
	VAR_IN_OUT
		aValue	:	TcVnVector2_REAL;	(* Value to set the container elements *)
	END_VAR
	VAR_INPUT
		hrPrev	:	HRESULT;	(* HRESULT indicating the result of previous operations (If SUCCEEDED(hrPrev) equals false, no operation is executed.) *)
	END_VAR

END_FUNCTION

// Functions/Basic Container Operations/F_VN_FillContainer/F_VN_FillContainer_TcVnVector2_SINT

	{attribute 'TcIecLibraryType'}
	{attribute 'external_name' := 'F_VN_FillContainer_TcVnVector2_SINT_GUID_755E5D68_48D3_2A88_5D5C_CB8922232F62'}
	(* Fill the container with the specified value. Only possible for containers with basic elements. *)
	FUNCTION F_VN_FillContainer_TcVnVector2_SINT : HRESULT
	VAR_INPUT
		ipContainer	:	ITcVnContainer;	(* Container with basic elements *)
	END_VAR
	VAR_IN_OUT
		aValue	:	TcVnVector2_SINT;	(* Value to set the container elements *)
	END_VAR
	VAR_INPUT
		hrPrev	:	HRESULT;	(* HRESULT indicating the result of previous operations (If SUCCEEDED(hrPrev) equals false, no operation is executed.) *)
	END_VAR

END_FUNCTION

// Functions/Basic Container Operations/F_VN_FillContainer/F_VN_FillContainer_TcVnVector2_UINT

	{attribute 'TcIecLibraryType'}
	{attribute 'external_name' := 'F_VN_FillContainer_TcVnVector2_UINT_GUID_F54099BC_053F_217E_6784_4C5ADAC0EC5F'}
	(* Fill the container with the specified value. Only possible for containers with basic elements. *)
	FUNCTION F_VN_FillContainer_TcVnVector2_UINT : HRESULT
	VAR_INPUT
		ipContainer	:	ITcVnContainer;	(* Container with basic elements *)
	END_VAR
	VAR_IN_OUT
		aValue	:	TcVnVector2_UINT;	(* Value to set the container elements *)
	END_VAR
	VAR_INPUT
		hrPrev	:	HRESULT;	(* HRESULT indicating the result of previous operations (If SUCCEEDED(hrPrev) equals false, no operation is executed.) *)
	END_VAR

END_FUNCTION

// Functions/Basic Container Operations/F_VN_FillContainer/F_VN_FillContainer_TcVnVector2_USINT

	{attribute 'TcIecLibraryType'}
	{attribute 'external_name' := 'F_VN_FillContainer_TcVnVector2_USINT_GUID_DD80526B_99D5_2FD7_6138_8477C955B2AF'}
	(* Fill the container with the specified value. Only possible for containers with basic elements. *)
	FUNCTION F_VN_FillContainer_TcVnVector2_USINT : HRESULT
	VAR_INPUT
		ipContainer	:	ITcVnContainer;	(* Container with basic elements *)
	END_VAR
	VAR_IN_OUT
		aValue	:	TcVnVector2_USINT;	(* Value to set the container elements *)
	END_VAR
	VAR_INPUT
		hrPrev	:	HRESULT;	(* HRESULT indicating the result of previous operations (If SUCCEEDED(hrPrev) equals false, no operation is executed.) *)
	END_VAR

END_FUNCTION

// Functions/Basic Container Operations/F_VN_FillContainer/F_VN_FillContainer_TcVnVector3_INT

	{attribute 'TcIecLibraryType'}
	{attribute 'external_name' := 'F_VN_FillContainer_TcVnVector3_INT_GUID_1E40EAB2_DB8D_2FCE_4F15_868BCA304DE8'}
	(* Fill the container with the specified value. Only possible for containers with basic elements. *)
	FUNCTION F_VN_FillContainer_TcVnVector3_INT : HRESULT
	VAR_INPUT
		ipContainer	:	ITcVnContainer;	(* Container with basic elements *)
	END_VAR
	VAR_IN_OUT
		aValue	:	TcVnVector3_INT;	(* Value to set the container elements *)
	END_VAR
	VAR_INPUT
		hrPrev	:	HRESULT;	(* HRESULT indicating the result of previous operations (If SUCCEEDED(hrPrev) equals false, no operation is executed.) *)
	END_VAR

END_FUNCTION

// Functions/Basic Container Operations/F_VN_FillContainer/F_VN_FillContainer_TcVnVector3_REAL

	{attribute 'TcIecLibraryType'}
	{attribute 'external_name' := 'F_VN_FillContainer_TcVnVector3_REAL_GUID_9B39B9A8_D00B_2C4B_772E_901B73B8543C'}
	(* Fill the container with the specified value. Only possible for containers with basic elements. *)
	FUNCTION F_VN_FillContainer_TcVnVector3_REAL : HRESULT
	VAR_INPUT
		ipContainer	:	ITcVnContainer;	(* Container with basic elements *)
	END_VAR
	VAR_IN_OUT
		aValue	:	TcVnVector3_REAL;	(* Value to set the container elements *)
	END_VAR
	VAR_INPUT
		hrPrev	:	HRESULT;	(* HRESULT indicating the result of previous operations (If SUCCEEDED(hrPrev) equals false, no operation is executed.) *)
	END_VAR

END_FUNCTION

// Functions/Basic Container Operations/F_VN_FillContainer/F_VN_FillContainer_TcVnVector3_SINT

	{attribute 'TcIecLibraryType'}
	{attribute 'external_name' := 'F_VN_FillContainer_TcVnVector3_SINT_GUID_72015BB1_0969_2729_6DC4_A789AC88E0F2'}
	(* Fill the container with the specified value. Only possible for containers with basic elements. *)
	FUNCTION F_VN_FillContainer_TcVnVector3_SINT : HRESULT
	VAR_INPUT
		ipContainer	:	ITcVnContainer;	(* Container with basic elements *)
	END_VAR
	VAR_IN_OUT
		aValue	:	TcVnVector3_SINT;	(* Value to set the container elements *)
	END_VAR
	VAR_INPUT
		hrPrev	:	HRESULT;	(* HRESULT indicating the result of previous operations (If SUCCEEDED(hrPrev) equals false, no operation is executed.) *)
	END_VAR

END_FUNCTION

// Functions/Basic Container Operations/F_VN_FillContainer/F_VN_FillContainer_TcVnVector3_UINT

	{attribute 'TcIecLibraryType'}
	{attribute 'external_name' := 'F_VN_FillContainer_TcVnVector3_UINT_GUID_4B6E421D_3CC0_2312_56AE_2EE386F16930'}
	(* Fill the container with the specified value. Only possible for containers with basic elements. *)
	FUNCTION F_VN_FillContainer_TcVnVector3_UINT : HRESULT
	VAR_INPUT
		ipContainer	:	ITcVnContainer;	(* Container with basic elements *)
	END_VAR
	VAR_IN_OUT
		aValue	:	TcVnVector3_UINT;	(* Value to set the container elements *)
	END_VAR
	VAR_INPUT
		hrPrev	:	HRESULT;	(* HRESULT indicating the result of previous operations (If SUCCEEDED(hrPrev) equals false, no operation is executed.) *)
	END_VAR

END_FUNCTION

// Functions/Basic Container Operations/F_VN_FillContainer/F_VN_FillContainer_TcVnVector3_USINT

	{attribute 'TcIecLibraryType'}
	{attribute 'external_name' := 'F_VN_FillContainer_TcVnVector3_USINT_GUID_2CF00519_00ED_2164_6F57_1F8CD7FD47FD'}
	(* Fill the container with the specified value. Only possible for containers with basic elements. *)
	FUNCTION F_VN_FillContainer_TcVnVector3_USINT : HRESULT
	VAR_INPUT
		ipContainer	:	ITcVnContainer;	(* Container with basic elements *)
	END_VAR
	VAR_IN_OUT
		aValue	:	TcVnVector3_USINT;	(* Value to set the container elements *)
	END_VAR
	VAR_INPUT
		hrPrev	:	HRESULT;	(* HRESULT indicating the result of previous operations (If SUCCEEDED(hrPrev) equals false, no operation is executed.) *)
	END_VAR

END_FUNCTION

// Functions/Basic Container Operations/F_VN_FillContainer/F_VN_FillContainer_TcVnVector4_DINT

	{attribute 'TcIecLibraryType'}
	{attribute 'external_name' := 'F_VN_FillContainer_TcVnVector4_DINT_GUID_94182C8B_6DDE_2B6B_517C_A260CECF94D3'}
	(* Fill the container with the specified value. Only possible for containers with basic elements. *)
	FUNCTION F_VN_FillContainer_TcVnVector4_DINT : HRESULT
	VAR_INPUT
		ipContainer	:	ITcVnContainer;	(* Container with basic elements *)
	END_VAR
	VAR_IN_OUT
		aValue	:	TcVnVector4_DINT;	(* Value to set the container elements *)
	END_VAR
	VAR_INPUT
		hrPrev	:	HRESULT;	(* HRESULT indicating the result of previous operations (If SUCCEEDED(hrPrev) equals false, no operation is executed.) *)
	END_VAR

END_FUNCTION

// Functions/Basic Container Operations/F_VN_FillContainer/F_VN_FillContainer_TcVnVector4_INT

	{attribute 'TcIecLibraryType'}
	{attribute 'external_name' := 'F_VN_FillContainer_TcVnVector4_INT_GUID_4AA9B3D2_9E42_2C83_404E_99FDE48AF550'}
	(* Fill the container with the specified value. Only possible for containers with basic elements. *)
	FUNCTION F_VN_FillContainer_TcVnVector4_INT : HRESULT
	VAR_INPUT
		ipContainer	:	ITcVnContainer;	(* Container with basic elements *)
	END_VAR
	VAR_IN_OUT
		aValue	:	TcVnVector4_INT;	(* Value to set the container elements *)
	END_VAR
	VAR_INPUT
		hrPrev	:	HRESULT;	(* HRESULT indicating the result of previous operations (If SUCCEEDED(hrPrev) equals false, no operation is executed.) *)
	END_VAR

END_FUNCTION

// Functions/Basic Container Operations/F_VN_FillContainer/F_VN_FillContainer_TcVnVector4_LREAL

	{attribute 'TcIecLibraryType'}
	{attribute 'external_name' := 'F_VN_FillContainer_TcVnVector4_LREAL_GUID_4D98B679_C8B1_2250_62B1_F8BE4BE660B7'}
	(* Fill the container with the specified value. Only possible for containers with basic elements. *)
	FUNCTION F_VN_FillContainer_TcVnVector4_LREAL : HRESULT
	VAR_INPUT
		ipContainer	:	ITcVnContainer;	(* Container with basic elements *)
	END_VAR
	VAR_IN_OUT
		aValue	:	TcVnVector4_LREAL;	(* Value to set the container elements *)
	END_VAR
	VAR_INPUT
		hrPrev	:	HRESULT;	(* HRESULT indicating the result of previous operations (If SUCCEEDED(hrPrev) equals false, no operation is executed.) *)
	END_VAR

END_FUNCTION

// Functions/Basic Container Operations/F_VN_FillContainer/F_VN_FillContainer_TcVnVector4_REAL

	{attribute 'TcIecLibraryType'}
	{attribute 'external_name' := 'F_VN_FillContainer_TcVnVector4_REAL_GUID_09724D77_A876_2B73_5394_820C4215AC68'}
	(* Fill the container with the specified value. Only possible for containers with basic elements. *)
	FUNCTION F_VN_FillContainer_TcVnVector4_REAL : HRESULT
	VAR_INPUT
		ipContainer	:	ITcVnContainer;	(* Container with basic elements *)
	END_VAR
	VAR_IN_OUT
		aValue	:	TcVnVector4_REAL;	(* Value to set the container elements *)
	END_VAR
	VAR_INPUT
		hrPrev	:	HRESULT;	(* HRESULT indicating the result of previous operations (If SUCCEEDED(hrPrev) equals false, no operation is executed.) *)
	END_VAR

END_FUNCTION

// Functions/Basic Container Operations/F_VN_FillContainer/F_VN_FillContainer_TcVnVector4_SINT

	{attribute 'TcIecLibraryType'}
	{attribute 'external_name' := 'F_VN_FillContainer_TcVnVector4_SINT_GUID_BE6A8137_521E_2F2C_47E1_AE05EA72FD60'}
	(* Fill the container with the specified value. Only possible for containers with basic elements. *)
	FUNCTION F_VN_FillContainer_TcVnVector4_SINT : HRESULT
	VAR_INPUT
		ipContainer	:	ITcVnContainer;	(* Container with basic elements *)
	END_VAR
	VAR_IN_OUT
		aValue	:	TcVnVector4_SINT;	(* Value to set the container elements *)
	END_VAR
	VAR_INPUT
		hrPrev	:	HRESULT;	(* HRESULT indicating the result of previous operations (If SUCCEEDED(hrPrev) equals false, no operation is executed.) *)
	END_VAR

END_FUNCTION

// Functions/Basic Container Operations/F_VN_FillContainer/F_VN_FillContainer_TcVnVector4_UINT

	{attribute 'TcIecLibraryType'}
	{attribute 'external_name' := 'F_VN_FillContainer_TcVnVector4_UINT_GUID_735A0BB6_DD5C_2B96_7147_6850719B1D2B'}
	(* Fill the container with the specified value. Only possible for containers with basic elements. *)
	FUNCTION F_VN_FillContainer_TcVnVector4_UINT : HRESULT
	VAR_INPUT
		ipContainer	:	ITcVnContainer;	(* Container with basic elements *)
	END_VAR
	VAR_IN_OUT
		aValue	:	TcVnVector4_UINT;	(* Value to set the container elements *)
	END_VAR
	VAR_INPUT
		hrPrev	:	HRESULT;	(* HRESULT indicating the result of previous operations (If SUCCEEDED(hrPrev) equals false, no operation is executed.) *)
	END_VAR

END_FUNCTION

// Functions/Basic Container Operations/F_VN_FillContainer/F_VN_FillContainer_TcVnVector4_USINT

	{attribute 'TcIecLibraryType'}
	{attribute 'external_name' := 'F_VN_FillContainer_TcVnVector4_USINT_GUID_A2A43896_463B_2FFD_5A18_9AE0A93BFF77'}
	(* Fill the container with the specified value. Only possible for containers with basic elements. *)
	FUNCTION F_VN_FillContainer_TcVnVector4_USINT : HRESULT
	VAR_INPUT
		ipContainer	:	ITcVnContainer;	(* Container with basic elements *)
	END_VAR
	VAR_IN_OUT
		aValue	:	TcVnVector4_USINT;	(* Value to set the container elements *)
	END_VAR
	VAR_INPUT
		hrPrev	:	HRESULT;	(* HRESULT indicating the result of previous operations (If SUCCEEDED(hrPrev) equals false, no operation is executed.) *)
	END_VAR

END_FUNCTION

// Functions/Basic Container Operations/F_VN_FillContainer/F_VN_FillContainer_UDINT

	{attribute 'TcIecLibraryType'}
	{attribute 'external_name' := 'F_VN_FillContainer_UDINT_GUID_239761D4_6171_2BF0_7B9C_090723BE5C16'}
	(* Fill the container with the specified value. Only possible for containers with basic elements. *)
	FUNCTION F_VN_FillContainer_UDINT : HRESULT
	VAR_INPUT
		ipContainer	:	ITcVnContainer;	(* Container with basic elements *)
		nValue	:	UDINT;	(* Value to set the container elements *)
		hrPrev	:	HRESULT;	(* HRESULT indicating the result of previous operations (If SUCCEEDED(hrPrev) equals false, no operation is executed.) *)
	END_VAR

END_FUNCTION

// Functions/Basic Container Operations/F_VN_FillContainer/F_VN_FillContainer_UINT

	{attribute 'TcIecLibraryType'}
	{attribute 'external_name' := 'F_VN_FillContainer_UINT_GUID_B5C8D570_00A0_2460_641D_7D9C83863B15'}
	(* Fill the container with the specified value. Only possible for containers with basic elements. *)
	FUNCTION F_VN_FillContainer_UINT : HRESULT
	VAR_INPUT
		ipContainer	:	ITcVnContainer;	(* Container with basic elements *)
		nValue	:	UINT;	(* Value to set the container elements *)
		hrPrev	:	HRESULT;	(* HRESULT indicating the result of previous operations (If SUCCEEDED(hrPrev) equals false, no operation is executed.) *)
	END_VAR

END_FUNCTION

// Functions/Basic Container Operations/F_VN_FillContainer/F_VN_FillContainer_ULINT

	{attribute 'TcIecLibraryType'}
	{attribute 'external_name' := 'F_VN_FillContainer_ULINT_GUID_1E1FF7E9_BDB2_2811_5F0B_2FDA5029F076'}
	(* Fill the container with the specified value. Only possible for containers with basic elements. *)
	FUNCTION F_VN_FillContainer_ULINT : HRESULT
	VAR_INPUT
		ipContainer	:	ITcVnContainer;	(* Container with basic elements *)
		nValue	:	ULINT;	(* Value to set the container elements *)
		hrPrev	:	HRESULT;	(* HRESULT indicating the result of previous operations (If SUCCEEDED(hrPrev) equals false, no operation is executed.) *)
	END_VAR

END_FUNCTION

// Functions/Basic Container Operations/F_VN_FillContainer/F_VN_FillContainer_USINT

	{attribute 'TcIecLibraryType'}
	{attribute 'external_name' := 'F_VN_FillContainer_USINT_GUID_74EFC9F2_240C_2D4E_5327_55DF9651E924'}
	(* Fill the container with the specified value. Only possible for containers with basic elements. *)
	FUNCTION F_VN_FillContainer_USINT : HRESULT
	VAR_INPUT
		ipContainer	:	ITcVnContainer;	(* Container with basic elements *)
		nValue	:	USINT;	(* Value to set the container elements *)
		hrPrev	:	HRESULT;	(* HRESULT indicating the result of previous operations (If SUCCEEDED(hrPrev) equals false, no operation is executed.) *)
	END_VAR

END_FUNCTION

// Functions/Basic Container Operations/F_VN_FillContainerExp/F_VN_FillContainerExp_DINT

	{attribute 'TcIecLibraryType'}
	{attribute 'external_name' := 'F_VN_FillContainerExp_DINT_GUID_CF7AE10F_AA4F_2A6A_5056_AF7AF6917B6C'}
	(* Partially fill the container with the specified value. Only possible for containers with basic elements. (expert function) *)
	FUNCTION F_VN_FillContainerExp_DINT : HRESULT
	VAR_INPUT
		ipContainer	:	ITcVnContainer;	(* Container with basic elements *)
		nValue	:	DINT;	(* Value to set the container elements *)
		nStartIdx	:	ULINT;	(* Start index *)
		nCount	:	ULINT;	(* Number of elements to set *)
		hrPrev	:	HRESULT;	(* HRESULT indicating the result of previous operations (If SUCCEEDED(hrPrev) equals false, no operation is executed.) *)
	END_VAR

END_FUNCTION

// Functions/Basic Container Operations/F_VN_FillContainerExp/F_VN_FillContainerExp_INT

	{attribute 'TcIecLibraryType'}
	{attribute 'external_name' := 'F_VN_FillContainerExp_INT_GUID_D4AB9897_D1AF_2C7F_4D0E_1667ED0662D8'}
	(* Partially fill the container with the specified value. Only possible for containers with basic elements. (expert function) *)
	FUNCTION F_VN_FillContainerExp_INT : HRESULT
	VAR_INPUT
		ipContainer	:	ITcVnContainer;	(* Container with basic elements *)
		nValue	:	INT;	(* Value to set the container elements *)
		nStartIdx	:	ULINT;	(* Start index *)
		nCount	:	ULINT;	(* Number of elements to set *)
		hrPrev	:	HRESULT;	(* HRESULT indicating the result of previous operations (If SUCCEEDED(hrPrev) equals false, no operation is executed.) *)
	END_VAR

END_FUNCTION

// Functions/Basic Container Operations/F_VN_FillContainerExp/F_VN_FillContainerExp_ITcVnImage

	{attribute 'TcIecLibraryType'}
	{attribute 'external_name' := 'F_VN_FillContainerExp_ITcVnImage_GUID_E1DE73EF_8B39_2828_4DE6_C97B3ADD179E'}
	(* Partially fill the container with the specified value. Only possible for containers with basic elements. (expert function) *)
	FUNCTION F_VN_FillContainerExp_ITcVnImage : HRESULT
	VAR_INPUT
		ipContainer	:	ITcVnContainer;	(* Container with basic elements *)
		ipValue	:	ITcVnImage;	(* Value to set the container elements *)
		nStartIdx	:	ULINT;	(* Start index *)
		nCount	:	ULINT;	(* Number of elements to set *)
		hrPrev	:	HRESULT;	(* HRESULT indicating the result of previous operations (If SUCCEEDED(hrPrev) equals false, no operation is executed.) *)
	END_VAR

END_FUNCTION

// Functions/Basic Container Operations/F_VN_FillContainerExp/F_VN_FillContainerExp_LREAL

	{attribute 'TcIecLibraryType'}
	{attribute 'external_name' := 'F_VN_FillContainerExp_LREAL_GUID_710575F2_B5A3_2483_5858_5F7523D1C9AA'}
	(* Partially fill the container with the specified value. Only possible for containers with basic elements. (expert function) *)
	FUNCTION F_VN_FillContainerExp_LREAL : HRESULT
	VAR_INPUT
		ipContainer	:	ITcVnContainer;	(* Container with basic elements *)
		fValue	:	LREAL;	(* Value to set the container elements *)
		nStartIdx	:	ULINT;	(* Start index *)
		nCount	:	ULINT;	(* Number of elements to set *)
		hrPrev	:	HRESULT;	(* HRESULT indicating the result of previous operations (If SUCCEEDED(hrPrev) equals false, no operation is executed.) *)
	END_VAR

END_FUNCTION

// Functions/Basic Container Operations/F_VN_FillContainerExp/F_VN_FillContainerExp_REAL

	{attribute 'TcIecLibraryType'}
	{attribute 'external_name' := 'F_VN_FillContainerExp_REAL_GUID_3F15C6E5_AF77_2749_689D_C88B9955B079'}
	(* Partially fill the container with the specified value. Only possible for containers with basic elements. (expert function) *)
	FUNCTION F_VN_FillContainerExp_REAL : HRESULT
	VAR_INPUT
		ipContainer	:	ITcVnContainer;	(* Container with basic elements *)
		fValue	:	REAL;	(* Value to set the container elements *)
		nStartIdx	:	ULINT;	(* Start index *)
		nCount	:	ULINT;	(* Number of elements to set *)
		hrPrev	:	HRESULT;	(* HRESULT indicating the result of previous operations (If SUCCEEDED(hrPrev) equals false, no operation is executed.) *)
	END_VAR

END_FUNCTION

// Functions/Basic Container Operations/F_VN_FillContainerExp/F_VN_FillContainerExp_SINT

	{attribute 'TcIecLibraryType'}
	{attribute 'external_name' := 'F_VN_FillContainerExp_SINT_GUID_E72BBCEE_2821_2A45_6269_7F97A882341D'}
	(* Partially fill the container with the specified value. Only possible for containers with basic elements. (expert function) *)
	FUNCTION F_VN_FillContainerExp_SINT : HRESULT
	VAR_INPUT
		ipContainer	:	ITcVnContainer;	(* Container with basic elements *)
		nValue	:	SINT;	(* Value to set the container elements *)
		nStartIdx	:	ULINT;	(* Start index *)
		nCount	:	ULINT;	(* Number of elements to set *)
		hrPrev	:	HRESULT;	(* HRESULT indicating the result of previous operations (If SUCCEEDED(hrPrev) equals false, no operation is executed.) *)
	END_VAR

END_FUNCTION

// Functions/Basic Container Operations/F_VN_FillContainerExp/F_VN_FillContainerExp_TcVnDMatch

	{attribute 'TcIecLibraryType'}
	{attribute 'external_name' := 'F_VN_FillContainerExp_TcVnDMatch_GUID_191EA90E_A049_2AC4_754C_A52535B28BAF'}
	(* Partially fill the container with the specified value. Only possible for containers with basic elements. (expert function) *)
	FUNCTION F_VN_FillContainerExp_TcVnDMatch : HRESULT
	VAR_INPUT
		ipContainer	:	ITcVnContainer;	(* Container with basic elements *)
	END_VAR
	VAR_IN_OUT
		stValue	:	TcVnDMatch;	(* Value to set the container elements *)
	END_VAR
	VAR_INPUT
		nStartIdx	:	ULINT;	(* Start index *)
		nCount	:	ULINT;	(* Number of elements to set *)
		hrPrev	:	HRESULT;	(* HRESULT indicating the result of previous operations (If SUCCEEDED(hrPrev) equals false, no operation is executed.) *)
	END_VAR

END_FUNCTION

// Functions/Basic Container Operations/F_VN_FillContainerExp/F_VN_FillContainerExp_TcVnKeyPoint

	{attribute 'TcIecLibraryType'}
	{attribute 'external_name' := 'F_VN_FillContainerExp_TcVnKeyPoint_GUID_292164B1_B67C_26F3_512F_C3463CC22C42'}
	(* Partially fill the container with the specified value. Only possible for containers with basic elements. (expert function) *)
	FUNCTION F_VN_FillContainerExp_TcVnKeyPoint : HRESULT
	VAR_INPUT
		ipContainer	:	ITcVnContainer;	(* Container with basic elements *)
	END_VAR
	VAR_IN_OUT
		stValue	:	TcVnKeyPoint;	(* Value to set the container elements *)
	END_VAR
	VAR_INPUT
		nStartIdx	:	ULINT;	(* Start index *)
		nCount	:	ULINT;	(* Number of elements to set *)
		hrPrev	:	HRESULT;	(* HRESULT indicating the result of previous operations (If SUCCEEDED(hrPrev) equals false, no operation is executed.) *)
	END_VAR

END_FUNCTION

// Functions/Basic Container Operations/F_VN_FillContainerExp/F_VN_FillContainerExp_TcVnPoint2_DINT

	{attribute 'TcIecLibraryType'}
	{attribute 'external_name' := 'F_VN_FillContainerExp_TcVnPoint2_DINT_GUID_225403B4_8E6C_2A81_4FA5_5B72291A5CA2'}
	(* Partially fill the container with the specified value. Only possible for containers with basic elements. (expert function) *)
	FUNCTION F_VN_FillContainerExp_TcVnPoint2_DINT : HRESULT
	VAR_INPUT
		ipContainer	:	ITcVnContainer;	(* Container with basic elements *)
	END_VAR
	VAR_IN_OUT
		aValue	:	TcVnPoint2_DINT;	(* Value to set the container elements *)
	END_VAR
	VAR_INPUT
		nStartIdx	:	ULINT;	(* Start index *)
		nCount	:	ULINT;	(* Number of elements to set *)
		hrPrev	:	HRESULT;	(* HRESULT indicating the result of previous operations (If SUCCEEDED(hrPrev) equals false, no operation is executed.) *)
	END_VAR

END_FUNCTION

// Functions/Basic Container Operations/F_VN_FillContainerExp/F_VN_FillContainerExp_TcVnPoint2_LREAL

	{attribute 'TcIecLibraryType'}
	{attribute 'external_name' := 'F_VN_FillContainerExp_TcVnPoint2_LREAL_GUID_985C30D8_69BE_2C55_7171_EA0EBAA40BB1'}
	(* Partially fill the container with the specified value. Only possible for containers with basic elements. (expert function) *)
	FUNCTION F_VN_FillContainerExp_TcVnPoint2_LREAL : HRESULT
	VAR_INPUT
		ipContainer	:	ITcVnContainer;	(* Container with basic elements *)
	END_VAR
	VAR_IN_OUT
		aValue	:	TcVnPoint2_LREAL;	(* Value to set the container elements *)
	END_VAR
	VAR_INPUT
		nStartIdx	:	ULINT;	(* Start index *)
		nCount	:	ULINT;	(* Number of elements to set *)
		hrPrev	:	HRESULT;	(* HRESULT indicating the result of previous operations (If SUCCEEDED(hrPrev) equals false, no operation is executed.) *)
	END_VAR

END_FUNCTION

// Functions/Basic Container Operations/F_VN_FillContainerExp/F_VN_FillContainerExp_TcVnPoint2_REAL

	{attribute 'TcIecLibraryType'}
	{attribute 'external_name' := 'F_VN_FillContainerExp_TcVnPoint2_REAL_GUID_A5389255_B367_29A0_7B59_2F8082E5234A'}
	(* Partially fill the container with the specified value. Only possible for containers with basic elements. (expert function) *)
	FUNCTION F_VN_FillContainerExp_TcVnPoint2_REAL : HRESULT
	VAR_INPUT
		ipContainer	:	ITcVnContainer;	(* Container with basic elements *)
	END_VAR
	VAR_IN_OUT
		aValue	:	TcVnPoint2_REAL;	(* Value to set the container elements *)
	END_VAR
	VAR_INPUT
		nStartIdx	:	ULINT;	(* Start index *)
		nCount	:	ULINT;	(* Number of elements to set *)
		hrPrev	:	HRESULT;	(* HRESULT indicating the result of previous operations (If SUCCEEDED(hrPrev) equals false, no operation is executed.) *)
	END_VAR

END_FUNCTION

// Functions/Basic Container Operations/F_VN_FillContainerExp/F_VN_FillContainerExp_TcVnPoint3_LREAL

	{attribute 'TcIecLibraryType'}
	{attribute 'external_name' := 'F_VN_FillContainerExp_TcVnPoint3_LREAL_GUID_C0C531B8_C514_2F84_6FBE_524EAEDB334F'}
	(* Partially fill the container with the specified value. Only possible for containers with basic elements. (expert function) *)
	FUNCTION F_VN_FillContainerExp_TcVnPoint3_LREAL : HRESULT
	VAR_INPUT
		ipContainer	:	ITcVnContainer;	(* Container with basic elements *)
	END_VAR
	VAR_IN_OUT
		aValue	:	TcVnPoint3_LREAL;	(* Value to set the container elements *)
	END_VAR
	VAR_INPUT
		nStartIdx	:	ULINT;	(* Start index *)
		nCount	:	ULINT;	(* Number of elements to set *)
		hrPrev	:	HRESULT;	(* HRESULT indicating the result of previous operations (If SUCCEEDED(hrPrev) equals false, no operation is executed.) *)
	END_VAR

END_FUNCTION

// Functions/Basic Container Operations/F_VN_FillContainerExp/F_VN_FillContainerExp_TcVnPoint3_REAL

	{attribute 'TcIecLibraryType'}
	{attribute 'external_name' := 'F_VN_FillContainerExp_TcVnPoint3_REAL_GUID_1D794A50_04CB_2FBA_6649_7F5B058D9189'}
	(* Partially fill the container with the specified value. Only possible for containers with basic elements. (expert function) *)
	FUNCTION F_VN_FillContainerExp_TcVnPoint3_REAL : HRESULT
	VAR_INPUT
		ipContainer	:	ITcVnContainer;	(* Container with basic elements *)
	END_VAR
	VAR_IN_OUT
		aValue	:	TcVnPoint3_REAL;	(* Value to set the container elements *)
	END_VAR
	VAR_INPUT
		nStartIdx	:	ULINT;	(* Start index *)
		nCount	:	ULINT;	(* Number of elements to set *)
		hrPrev	:	HRESULT;	(* HRESULT indicating the result of previous operations (If SUCCEEDED(hrPrev) equals false, no operation is executed.) *)
	END_VAR

END_FUNCTION

// Functions/Basic Container Operations/F_VN_FillContainerExp/F_VN_FillContainerExp_TcVnRectangle_DINT

	{attribute 'TcIecLibraryType'}
	{attribute 'external_name' := 'F_VN_FillContainerExp_TcVnRectangle_DINT_GUID_FC11ABB9_5419_29A8_61C3_17D524DCA8C2'}
	(* Partially fill the container with the specified value. Only possible for containers with basic elements. (expert function) *)
	FUNCTION F_VN_FillContainerExp_TcVnRectangle_DINT : HRESULT
	VAR_INPUT
		ipContainer	:	ITcVnContainer;	(* Container with basic elements *)
	END_VAR
	VAR_IN_OUT
		stValue	:	TcVnRectangle_DINT;	(* Value to set the container elements *)
	END_VAR
	VAR_INPUT
		nStartIdx	:	ULINT;	(* Start index *)
		nCount	:	ULINT;	(* Number of elements to set *)
		hrPrev	:	HRESULT;	(* HRESULT indicating the result of previous operations (If SUCCEEDED(hrPrev) equals false, no operation is executed.) *)
	END_VAR

END_FUNCTION

// Functions/Basic Container Operations/F_VN_FillContainerExp/F_VN_FillContainerExp_TcVnRotatedRectangle

	{attribute 'TcIecLibraryType'}
	{attribute 'external_name' := 'F_VN_FillContainerExp_TcVnRotatedRectangle_GUID_2FCAA197_9E65_2484_56D5_0AAEAC15979B'}
	(* Partially fill the container with the specified value. Only possible for containers with basic elements. (expert function) *)
	FUNCTION F_VN_FillContainerExp_TcVnRotatedRectangle : HRESULT
	VAR_INPUT
		ipContainer	:	ITcVnContainer;	(* Container with basic elements *)
	END_VAR
	VAR_IN_OUT
		stValue	:	TcVnRotatedRectangle;	(* Value to set the container elements *)
	END_VAR
	VAR_INPUT
		nStartIdx	:	ULINT;	(* Start index *)
		nCount	:	ULINT;	(* Number of elements to set *)
		hrPrev	:	HRESULT;	(* HRESULT indicating the result of previous operations (If SUCCEEDED(hrPrev) equals false, no operation is executed.) *)
	END_VAR

END_FUNCTION

// Functions/Basic Container Operations/F_VN_FillContainerExp/F_VN_FillContainerExp_TcVnVector2_DINT

	{attribute 'TcIecLibraryType'}
	{attribute 'external_name' := 'F_VN_FillContainerExp_TcVnVector2_DINT_GUID_A283EB52_EE86_2B1B_7467_B6FDB850F1BB'}
	(* Partially fill the container with the specified value. Only possible for containers with basic elements. (expert function) *)
	FUNCTION F_VN_FillContainerExp_TcVnVector2_DINT : HRESULT
	VAR_INPUT
		ipContainer	:	ITcVnContainer;	(* Container with basic elements *)
	END_VAR
	VAR_IN_OUT
		aValue	:	TcVnVector2_DINT;	(* Value to set the container elements *)
	END_VAR
	VAR_INPUT
		nStartIdx	:	ULINT;	(* Start index *)
		nCount	:	ULINT;	(* Number of elements to set *)
		hrPrev	:	HRESULT;	(* HRESULT indicating the result of previous operations (If SUCCEEDED(hrPrev) equals false, no operation is executed.) *)
	END_VAR

END_FUNCTION

// Functions/Basic Container Operations/F_VN_FillContainerExp/F_VN_FillContainerExp_TcVnVector2_INT

	{attribute 'TcIecLibraryType'}
	{attribute 'external_name' := 'F_VN_FillContainerExp_TcVnVector2_INT_GUID_8706F0BC_CEFC_2223_4380_68B41C6E5B25'}
	(* Partially fill the container with the specified value. Only possible for containers with basic elements. (expert function) *)
	FUNCTION F_VN_FillContainerExp_TcVnVector2_INT : HRESULT
	VAR_INPUT
		ipContainer	:	ITcVnContainer;	(* Container with basic elements *)
	END_VAR
	VAR_IN_OUT
		aValue	:	TcVnVector2_INT;	(* Value to set the container elements *)
	END_VAR
	VAR_INPUT
		nStartIdx	:	ULINT;	(* Start index *)
		nCount	:	ULINT;	(* Number of elements to set *)
		hrPrev	:	HRESULT;	(* HRESULT indicating the result of previous operations (If SUCCEEDED(hrPrev) equals false, no operation is executed.) *)
	END_VAR

END_FUNCTION

// Functions/Basic Container Operations/F_VN_FillContainerExp/F_VN_FillContainerExp_TcVnVector2_REAL

	{attribute 'TcIecLibraryType'}
	{attribute 'external_name' := 'F_VN_FillContainerExp_TcVnVector2_REAL_GUID_0E7E6CB5_E97F_2BEB_4398_9AE29D2D1D97'}
	(* Partially fill the container with the specified value. Only possible for containers with basic elements. (expert function) *)
	FUNCTION F_VN_FillContainerExp_TcVnVector2_REAL : HRESULT
	VAR_INPUT
		ipContainer	:	ITcVnContainer;	(* Container with basic elements *)
	END_VAR
	VAR_IN_OUT
		aValue	:	TcVnVector2_REAL;	(* Value to set the container elements *)
	END_VAR
	VAR_INPUT
		nStartIdx	:	ULINT;	(* Start index *)
		nCount	:	ULINT;	(* Number of elements to set *)
		hrPrev	:	HRESULT;	(* HRESULT indicating the result of previous operations (If SUCCEEDED(hrPrev) equals false, no operation is executed.) *)
	END_VAR

END_FUNCTION

// Functions/Basic Container Operations/F_VN_FillContainerExp/F_VN_FillContainerExp_TcVnVector2_SINT

	{attribute 'TcIecLibraryType'}
	{attribute 'external_name' := 'F_VN_FillContainerExp_TcVnVector2_SINT_GUID_2DCDEE71_C1E8_2E15_64CA_5570500E79EB'}
	(* Partially fill the container with the specified value. Only possible for containers with basic elements. (expert function) *)
	FUNCTION F_VN_FillContainerExp_TcVnVector2_SINT : HRESULT
	VAR_INPUT
		ipContainer	:	ITcVnContainer;	(* Container with basic elements *)
	END_VAR
	VAR_IN_OUT
		aValue	:	TcVnVector2_SINT;	(* Value to set the container elements *)
	END_VAR
	VAR_INPUT
		nStartIdx	:	ULINT;	(* Start index *)
		nCount	:	ULINT;	(* Number of elements to set *)
		hrPrev	:	HRESULT;	(* HRESULT indicating the result of previous operations (If SUCCEEDED(hrPrev) equals false, no operation is executed.) *)
	END_VAR

END_FUNCTION

// Functions/Basic Container Operations/F_VN_FillContainerExp/F_VN_FillContainerExp_TcVnVector2_UINT

	{attribute 'TcIecLibraryType'}
	{attribute 'external_name' := 'F_VN_FillContainerExp_TcVnVector2_UINT_GUID_5F7A601B_B98D_2BFE_5755_F74C9599F32B'}
	(* Partially fill the container with the specified value. Only possible for containers with basic elements. (expert function) *)
	FUNCTION F_VN_FillContainerExp_TcVnVector2_UINT : HRESULT
	VAR_INPUT
		ipContainer	:	ITcVnContainer;	(* Container with basic elements *)
	END_VAR
	VAR_IN_OUT
		aValue	:	TcVnVector2_UINT;	(* Value to set the container elements *)
	END_VAR
	VAR_INPUT
		nStartIdx	:	ULINT;	(* Start index *)
		nCount	:	ULINT;	(* Number of elements to set *)
		hrPrev	:	HRESULT;	(* HRESULT indicating the result of previous operations (If SUCCEEDED(hrPrev) equals false, no operation is executed.) *)
	END_VAR

END_FUNCTION

// Functions/Basic Container Operations/F_VN_FillContainerExp/F_VN_FillContainerExp_TcVnVector2_USINT

	{attribute 'TcIecLibraryType'}
	{attribute 'external_name' := 'F_VN_FillContainerExp_TcVnVector2_USINT_GUID_BD73CC2F_D28F_2C26_4947_CDEA4EAFA5D3'}
	(* Partially fill the container with the specified value. Only possible for containers with basic elements. (expert function) *)
	FUNCTION F_VN_FillContainerExp_TcVnVector2_USINT : HRESULT
	VAR_INPUT
		ipContainer	:	ITcVnContainer;	(* Container with basic elements *)
	END_VAR
	VAR_IN_OUT
		aValue	:	TcVnVector2_USINT;	(* Value to set the container elements *)
	END_VAR
	VAR_INPUT
		nStartIdx	:	ULINT;	(* Start index *)
		nCount	:	ULINT;	(* Number of elements to set *)
		hrPrev	:	HRESULT;	(* HRESULT indicating the result of previous operations (If SUCCEEDED(hrPrev) equals false, no operation is executed.) *)
	END_VAR

END_FUNCTION

// Functions/Basic Container Operations/F_VN_FillContainerExp/F_VN_FillContainerExp_TcVnVector3_INT

	{attribute 'TcIecLibraryType'}
	{attribute 'external_name' := 'F_VN_FillContainerExp_TcVnVector3_INT_GUID_FFDFE8EC_BB9A_2BFD_69E7_438438F71696'}
	(* Partially fill the container with the specified value. Only possible for containers with basic elements. (expert function) *)
	FUNCTION F_VN_FillContainerExp_TcVnVector3_INT : HRESULT
	VAR_INPUT
		ipContainer	:	ITcVnContainer;	(* Container with basic elements *)
	END_VAR
	VAR_IN_OUT
		aValue	:	TcVnVector3_INT;	(* Value to set the container elements *)
	END_VAR
	VAR_INPUT
		nStartIdx	:	ULINT;	(* Start index *)
		nCount	:	ULINT;	(* Number of elements to set *)
		hrPrev	:	HRESULT;	(* HRESULT indicating the result of previous operations (If SUCCEEDED(hrPrev) equals false, no operation is executed.) *)
	END_VAR

END_FUNCTION

// Functions/Basic Container Operations/F_VN_FillContainerExp/F_VN_FillContainerExp_TcVnVector3_REAL

	{attribute 'TcIecLibraryType'}
	{attribute 'external_name' := 'F_VN_FillContainerExp_TcVnVector3_REAL_GUID_80B38832_6FEC_25AD_476F_F4EA56A4DCC3'}
	(* Partially fill the container with the specified value. Only possible for containers with basic elements. (expert function) *)
	FUNCTION F_VN_FillContainerExp_TcVnVector3_REAL : HRESULT
	VAR_INPUT
		ipContainer	:	ITcVnContainer;	(* Container with basic elements *)
	END_VAR
	VAR_IN_OUT
		aValue	:	TcVnVector3_REAL;	(* Value to set the container elements *)
	END_VAR
	VAR_INPUT
		nStartIdx	:	ULINT;	(* Start index *)
		nCount	:	ULINT;	(* Number of elements to set *)
		hrPrev	:	HRESULT;	(* HRESULT indicating the result of previous operations (If SUCCEEDED(hrPrev) equals false, no operation is executed.) *)
	END_VAR

END_FUNCTION

// Functions/Basic Container Operations/F_VN_FillContainerExp/F_VN_FillContainerExp_TcVnVector3_SINT

	{attribute 'TcIecLibraryType'}
	{attribute 'external_name' := 'F_VN_FillContainerExp_TcVnVector3_SINT_GUID_B0CA3E98_B115_293A_5075_4C46EFBF7EA5'}
	(* Partially fill the container with the specified value. Only possible for containers with basic elements. (expert function) *)
	FUNCTION F_VN_FillContainerExp_TcVnVector3_SINT : HRESULT
	VAR_INPUT
		ipContainer	:	ITcVnContainer;	(* Container with basic elements *)
	END_VAR
	VAR_IN_OUT
		aValue	:	TcVnVector3_SINT;	(* Value to set the container elements *)
	END_VAR
	VAR_INPUT
		nStartIdx	:	ULINT;	(* Start index *)
		nCount	:	ULINT;	(* Number of elements to set *)
		hrPrev	:	HRESULT;	(* HRESULT indicating the result of previous operations (If SUCCEEDED(hrPrev) equals false, no operation is executed.) *)
	END_VAR

END_FUNCTION

// Functions/Basic Container Operations/F_VN_FillContainerExp/F_VN_FillContainerExp_TcVnVector3_UINT

	{attribute 'TcIecLibraryType'}
	{attribute 'external_name' := 'F_VN_FillContainerExp_TcVnVector3_UINT_GUID_D59F44A0_0DC1_24F5_5FEA_77097D8B4574'}
	(* Partially fill the container with the specified value. Only possible for containers with basic elements. (expert function) *)
	FUNCTION F_VN_FillContainerExp_TcVnVector3_UINT : HRESULT
	VAR_INPUT
		ipContainer	:	ITcVnContainer;	(* Container with basic elements *)
	END_VAR
	VAR_IN_OUT
		aValue	:	TcVnVector3_UINT;	(* Value to set the container elements *)
	END_VAR
	VAR_INPUT
		nStartIdx	:	ULINT;	(* Start index *)
		nCount	:	ULINT;	(* Number of elements to set *)
		hrPrev	:	HRESULT;	(* HRESULT indicating the result of previous operations (If SUCCEEDED(hrPrev) equals false, no operation is executed.) *)
	END_VAR

END_FUNCTION

// Functions/Basic Container Operations/F_VN_FillContainerExp/F_VN_FillContainerExp_TcVnVector3_USINT

	{attribute 'TcIecLibraryType'}
	{attribute 'external_name' := 'F_VN_FillContainerExp_TcVnVector3_USINT_GUID_D8DA6202_56E9_2E36_7653_AD6D88C2884B'}
	(* Partially fill the container with the specified value. Only possible for containers with basic elements. (expert function) *)
	FUNCTION F_VN_FillContainerExp_TcVnVector3_USINT : HRESULT
	VAR_INPUT
		ipContainer	:	ITcVnContainer;	(* Container with basic elements *)
	END_VAR
	VAR_IN_OUT
		aValue	:	TcVnVector3_USINT;	(* Value to set the container elements *)
	END_VAR
	VAR_INPUT
		nStartIdx	:	ULINT;	(* Start index *)
		nCount	:	ULINT;	(* Number of elements to set *)
		hrPrev	:	HRESULT;	(* HRESULT indicating the result of previous operations (If SUCCEEDED(hrPrev) equals false, no operation is executed.) *)
	END_VAR

END_FUNCTION

// Functions/Basic Container Operations/F_VN_FillContainerExp/F_VN_FillContainerExp_TcVnVector4_DINT

	{attribute 'TcIecLibraryType'}
	{attribute 'external_name' := 'F_VN_FillContainerExp_TcVnVector4_DINT_GUID_A719F079_E06D_2EDD_4A11_4B43DA7038B2'}
	(* Partially fill the container with the specified value. Only possible for containers with basic elements. (expert function) *)
	FUNCTION F_VN_FillContainerExp_TcVnVector4_DINT : HRESULT
	VAR_INPUT
		ipContainer	:	ITcVnContainer;	(* Container with basic elements *)
	END_VAR
	VAR_IN_OUT
		aValue	:	TcVnVector4_DINT;	(* Value to set the container elements *)
	END_VAR
	VAR_INPUT
		nStartIdx	:	ULINT;	(* Start index *)
		nCount	:	ULINT;	(* Number of elements to set *)
		hrPrev	:	HRESULT;	(* HRESULT indicating the result of previous operations (If SUCCEEDED(hrPrev) equals false, no operation is executed.) *)
	END_VAR

END_FUNCTION

// Functions/Basic Container Operations/F_VN_FillContainerExp/F_VN_FillContainerExp_TcVnVector4_INT

	{attribute 'TcIecLibraryType'}
	{attribute 'external_name' := 'F_VN_FillContainerExp_TcVnVector4_INT_GUID_89AA5534_1B75_29F2_6139_808DCAA157DF'}
	(* Partially fill the container with the specified value. Only possible for containers with basic elements. (expert function) *)
	FUNCTION F_VN_FillContainerExp_TcVnVector4_INT : HRESULT
	VAR_INPUT
		ipContainer	:	ITcVnContainer;	(* Container with basic elements *)
	END_VAR
	VAR_IN_OUT
		aValue	:	TcVnVector4_INT;	(* Value to set the container elements *)
	END_VAR
	VAR_INPUT
		nStartIdx	:	ULINT;	(* Start index *)
		nCount	:	ULINT;	(* Number of elements to set *)
		hrPrev	:	HRESULT;	(* HRESULT indicating the result of previous operations (If SUCCEEDED(hrPrev) equals false, no operation is executed.) *)
	END_VAR

END_FUNCTION

// Functions/Basic Container Operations/F_VN_FillContainerExp/F_VN_FillContainerExp_TcVnVector4_LREAL

	{attribute 'TcIecLibraryType'}
	{attribute 'external_name' := 'F_VN_FillContainerExp_TcVnVector4_LREAL_GUID_A93CF1EE_D88B_2621_5AD0_A2F95ED40D60'}
	(* Partially fill the container with the specified value. Only possible for containers with basic elements. (expert function) *)
	FUNCTION F_VN_FillContainerExp_TcVnVector4_LREAL : HRESULT
	VAR_INPUT
		ipContainer	:	ITcVnContainer;	(* Container with basic elements *)
	END_VAR
	VAR_IN_OUT
		aValue	:	TcVnVector4_LREAL;	(* Value to set the container elements *)
	END_VAR
	VAR_INPUT
		nStartIdx	:	ULINT;	(* Start index *)
		nCount	:	ULINT;	(* Number of elements to set *)
		hrPrev	:	HRESULT;	(* HRESULT indicating the result of previous operations (If SUCCEEDED(hrPrev) equals false, no operation is executed.) *)
	END_VAR

END_FUNCTION

// Functions/Basic Container Operations/F_VN_FillContainerExp/F_VN_FillContainerExp_TcVnVector4_REAL

	{attribute 'TcIecLibraryType'}
	{attribute 'external_name' := 'F_VN_FillContainerExp_TcVnVector4_REAL_GUID_9A249C43_266C_2BBA_7135_10AC0DD7842C'}
	(* Partially fill the container with the specified value. Only possible for containers with basic elements. (expert function) *)
	FUNCTION F_VN_FillContainerExp_TcVnVector4_REAL : HRESULT
	VAR_INPUT
		ipContainer	:	ITcVnContainer;	(* Container with basic elements *)
	END_VAR
	VAR_IN_OUT
		aValue	:	TcVnVector4_REAL;	(* Value to set the container elements *)
	END_VAR
	VAR_INPUT
		nStartIdx	:	ULINT;	(* Start index *)
		nCount	:	ULINT;	(* Number of elements to set *)
		hrPrev	:	HRESULT;	(* HRESULT indicating the result of previous operations (If SUCCEEDED(hrPrev) equals false, no operation is executed.) *)
	END_VAR

END_FUNCTION

// Functions/Basic Container Operations/F_VN_FillContainerExp/F_VN_FillContainerExp_TcVnVector4_SINT

	{attribute 'TcIecLibraryType'}
	{attribute 'external_name' := 'F_VN_FillContainerExp_TcVnVector4_SINT_GUID_4102C419_AE30_2BC5_6EAE_5B026E2B8193'}
	(* Partially fill the container with the specified value. Only possible for containers with basic elements. (expert function) *)
	FUNCTION F_VN_FillContainerExp_TcVnVector4_SINT : HRESULT
	VAR_INPUT
		ipContainer	:	ITcVnContainer;	(* Container with basic elements *)
	END_VAR
	VAR_IN_OUT
		aValue	:	TcVnVector4_SINT;	(* Value to set the container elements *)
	END_VAR
	VAR_INPUT
		nStartIdx	:	ULINT;	(* Start index *)
		nCount	:	ULINT;	(* Number of elements to set *)
		hrPrev	:	HRESULT;	(* HRESULT indicating the result of previous operations (If SUCCEEDED(hrPrev) equals false, no operation is executed.) *)
	END_VAR

END_FUNCTION

// Functions/Basic Container Operations/F_VN_FillContainerExp/F_VN_FillContainerExp_TcVnVector4_UINT

	{attribute 'TcIecLibraryType'}
	{attribute 'external_name' := 'F_VN_FillContainerExp_TcVnVector4_UINT_GUID_18AFDAD2_2497_2E70_4906_EC40F561003F'}
	(* Partially fill the container with the specified value. Only possible for containers with basic elements. (expert function) *)
	FUNCTION F_VN_FillContainerExp_TcVnVector4_UINT : HRESULT
	VAR_INPUT
		ipContainer	:	ITcVnContainer;	(* Container with basic elements *)
	END_VAR
	VAR_IN_OUT
		aValue	:	TcVnVector4_UINT;	(* Value to set the container elements *)
	END_VAR
	VAR_INPUT
		nStartIdx	:	ULINT;	(* Start index *)
		nCount	:	ULINT;	(* Number of elements to set *)
		hrPrev	:	HRESULT;	(* HRESULT indicating the result of previous operations (If SUCCEEDED(hrPrev) equals false, no operation is executed.) *)
	END_VAR

END_FUNCTION

// Functions/Basic Container Operations/F_VN_FillContainerExp/F_VN_FillContainerExp_TcVnVector4_USINT

	{attribute 'TcIecLibraryType'}
	{attribute 'external_name' := 'F_VN_FillContainerExp_TcVnVector4_USINT_GUID_FF5B9C1F_2DE4_231F_572D_3FA0550EDDD3'}
	(* Partially fill the container with the specified value. Only possible for containers with basic elements. (expert function) *)
	FUNCTION F_VN_FillContainerExp_TcVnVector4_USINT : HRESULT
	VAR_INPUT
		ipContainer	:	ITcVnContainer;	(* Container with basic elements *)
	END_VAR
	VAR_IN_OUT
		aValue	:	TcVnVector4_USINT;	(* Value to set the container elements *)
	END_VAR
	VAR_INPUT
		nStartIdx	:	ULINT;	(* Start index *)
		nCount	:	ULINT;	(* Number of elements to set *)
		hrPrev	:	HRESULT;	(* HRESULT indicating the result of previous operations (If SUCCEEDED(hrPrev) equals false, no operation is executed.) *)
	END_VAR

END_FUNCTION

// Functions/Basic Container Operations/F_VN_FillContainerExp/F_VN_FillContainerExp_UDINT

	{attribute 'TcIecLibraryType'}
	{attribute 'external_name' := 'F_VN_FillContainerExp_UDINT_GUID_B6241AFA_BEC0_2A05_4054_04AA25F39C43'}
	(* Partially fill the container with the specified value. Only possible for containers with basic elements. (expert function) *)
	FUNCTION F_VN_FillContainerExp_UDINT : HRESULT
	VAR_INPUT
		ipContainer	:	ITcVnContainer;	(* Container with basic elements *)
		nValue	:	UDINT;	(* Value to set the container elements *)
		nStartIdx	:	ULINT;	(* Start index *)
		nCount	:	ULINT;	(* Number of elements to set *)
		hrPrev	:	HRESULT;	(* HRESULT indicating the result of previous operations (If SUCCEEDED(hrPrev) equals false, no operation is executed.) *)
	END_VAR

END_FUNCTION

// Functions/Basic Container Operations/F_VN_FillContainerExp/F_VN_FillContainerExp_UINT

	{attribute 'TcIecLibraryType'}
	{attribute 'external_name' := 'F_VN_FillContainerExp_UINT_GUID_318851FA_AD3E_2646_7225_CA6BD4299F2C'}
	(* Partially fill the container with the specified value. Only possible for containers with basic elements. (expert function) *)
	FUNCTION F_VN_FillContainerExp_UINT : HRESULT
	VAR_INPUT
		ipContainer	:	ITcVnContainer;	(* Container with basic elements *)
		nValue	:	UINT;	(* Value to set the container elements *)
		nStartIdx	:	ULINT;	(* Start index *)
		nCount	:	ULINT;	(* Number of elements to set *)
		hrPrev	:	HRESULT;	(* HRESULT indicating the result of previous operations (If SUCCEEDED(hrPrev) equals false, no operation is executed.) *)
	END_VAR

END_FUNCTION

// Functions/Basic Container Operations/F_VN_FillContainerExp/F_VN_FillContainerExp_ULINT

	{attribute 'TcIecLibraryType'}
	{attribute 'external_name' := 'F_VN_FillContainerExp_ULINT_GUID_96FA93D5_FE80_2B56_418F_4817CC6692D9'}
	(* Partially fill the container with the specified value. Only possible for containers with basic elements. (expert function) *)
	FUNCTION F_VN_FillContainerExp_ULINT : HRESULT
	VAR_INPUT
		ipContainer	:	ITcVnContainer;	(* Container with basic elements *)
		nValue	:	ULINT;	(* Value to set the container elements *)
		nStartIdx	:	ULINT;	(* Start index *)
		nCount	:	ULINT;	(* Number of elements to set *)
		hrPrev	:	HRESULT;	(* HRESULT indicating the result of previous operations (If SUCCEEDED(hrPrev) equals false, no operation is executed.) *)
	END_VAR

END_FUNCTION

// Functions/Basic Container Operations/F_VN_FillContainerExp/F_VN_FillContainerExp_USINT

	{attribute 'TcIecLibraryType'}
	{attribute 'external_name' := 'F_VN_FillContainerExp_USINT_GUID_294399BB_17B3_2497_59A4_F0C3BBC36F13'}
	(* Partially fill the container with the specified value. Only possible for containers with basic elements. (expert function) *)
	FUNCTION F_VN_FillContainerExp_USINT : HRESULT
	VAR_INPUT
		ipContainer	:	ITcVnContainer;	(* Container with basic elements *)
		nValue	:	USINT;	(* Value to set the container elements *)
		nStartIdx	:	ULINT;	(* Start index *)
		nCount	:	ULINT;	(* Number of elements to set *)
		hrPrev	:	HRESULT;	(* HRESULT indicating the result of previous operations (If SUCCEEDED(hrPrev) equals false, no operation is executed.) *)
	END_VAR

END_FUNCTION

// Functions/Basic Container Operations/F_VN_GetAt/F_VN_GetAt_ITcVnContainer

	{attribute 'TcIecLibraryType'}
	{attribute 'external_name' := 'F_VN_GetAt_ITcVnContainer_GUID_73F234EF_EC9A_2955_5AE0_AC2AE38956ED'}
	(* Gets the ITcVnContainer element at the specified index of the source container. (Alternatively use interface method .GetAt.) *)
	FUNCTION F_VN_GetAt_ITcVnContainer : HRESULT
	VAR_INPUT
		ipSrcContainer	:	ITcVnContainer;	(* Container with ITcVnContainer elements *)
		ipDestContainer	:	REFERENCE TO ITcVnContainer;	(* Returns the container at the specified index *)
		nIndex	:	ULINT;	(* Index of the requested element *)
		hrPrev	:	HRESULT;	(* HRESULT indicating the result of previous operations (If SUCCEEDED(hrPrev) equals false, no operation is executed.) *)
	END_VAR

END_FUNCTION

// Functions/Basic Container Operations/F_VN_GetAt/F_VN_GetAt_DINT

	{attribute 'TcIecLibraryType'}
	{attribute 'external_name' := 'F_VN_GetAt_DINT_GUID_A454BB75_2430_2E40_71DB_8A43D2BD9060'}
	(* Gets the DINT element at the specified index of the container. *)
	FUNCTION F_VN_GetAt_DINT : HRESULT
	VAR_INPUT
		ipContainer	:	ITcVnContainer;	(* Container with DINT elements *)
	END_VAR
	VAR_IN_OUT
		nElement	:	DINT;	(* Returns the element at the specified index *)
	END_VAR
	VAR_INPUT
		nIndex	:	ULINT;	(* Index of the requested element *)
		hrPrev	:	HRESULT;	(* HRESULT indicating the result of previous operations (If SUCCEEDED(hrPrev) equals false, no operation is executed.) *)
	END_VAR

END_FUNCTION

// Functions/Basic Container Operations/F_VN_GetAt/F_VN_GetAt_INT

	{attribute 'TcIecLibraryType'}
	{attribute 'external_name' := 'F_VN_GetAt_INT_GUID_EC2EC01B_1ECF_24E9_5960_266768271925'}
	(* Gets the INT element at the specified index of the container. *)
	FUNCTION F_VN_GetAt_INT : HRESULT
	VAR_INPUT
		ipContainer	:	ITcVnContainer;	(* Container with INT elements *)
	END_VAR
	VAR_IN_OUT
		nElement	:	INT;	(* Returns the element at the specified index *)
	END_VAR
	VAR_INPUT
		nIndex	:	ULINT;	(* Index of the requested element *)
		hrPrev	:	HRESULT;	(* HRESULT indicating the result of previous operations (If SUCCEEDED(hrPrev) equals false, no operation is executed.) *)
	END_VAR

END_FUNCTION

// Functions/Basic Container Operations/F_VN_GetAt/F_VN_GetAt_ITcVnImage

	{attribute 'TcIecLibraryType'}
	{attribute 'external_name' := 'F_VN_GetAt_ITcVnImage_GUID_EB3BF424_C86C_2C12_5F0A_76B3988F393D'}
	(* Gets the ITcVnImage element at the specified index of the container. *)
	FUNCTION F_VN_GetAt_ITcVnImage : HRESULT
	VAR_INPUT
		ipContainer	:	ITcVnContainer;	(* Container with ITcVnImage elements *)
		ipElement	:	REFERENCE TO ITcVnImage;	(* Returns the element at the specified index *)
		nIndex	:	ULINT;	(* Index of the requested element *)
		hrPrev	:	HRESULT;	(* HRESULT indicating the result of previous operations (If SUCCEEDED(hrPrev) equals false, no operation is executed.) *)
	END_VAR

END_FUNCTION

// Functions/Basic Container Operations/F_VN_GetAt/F_VN_GetAt_LREAL

	{attribute 'TcIecLibraryType'}
	{attribute 'external_name' := 'F_VN_GetAt_LREAL_GUID_AB2AEB47_987A_2B14_6052_4C0EF7972EC5'}
	(* Gets the LREAL element at the specified index of the container. *)
	FUNCTION F_VN_GetAt_LREAL : HRESULT
	VAR_INPUT
		ipContainer	:	ITcVnContainer;	(* Container with LREAL elements *)
	END_VAR
	VAR_IN_OUT
		fElement	:	LREAL;	(* Returns the element at the specified index *)
	END_VAR
	VAR_INPUT
		nIndex	:	ULINT;	(* Index of the requested element *)
		hrPrev	:	HRESULT;	(* HRESULT indicating the result of previous operations (If SUCCEEDED(hrPrev) equals false, no operation is executed.) *)
	END_VAR

END_FUNCTION

// Functions/Basic Container Operations/F_VN_GetAt/F_VN_GetAt_REAL

	{attribute 'TcIecLibraryType'}
	{attribute 'external_name' := 'F_VN_GetAt_REAL_GUID_69BB15FA_CB11_2E1B_7611_9DF69206E027'}
	(* Gets the REAL element at the specified index of the container. *)
	FUNCTION F_VN_GetAt_REAL : HRESULT
	VAR_INPUT
		ipContainer	:	ITcVnContainer;	(* Container with REAL elements *)
	END_VAR
	VAR_IN_OUT
		fElement	:	REAL;	(* Returns the element at the specified index *)
	END_VAR
	VAR_INPUT
		nIndex	:	ULINT;	(* Index of the requested element *)
		hrPrev	:	HRESULT;	(* HRESULT indicating the result of previous operations (If SUCCEEDED(hrPrev) equals false, no operation is executed.) *)
	END_VAR

END_FUNCTION

// Functions/Basic Container Operations/F_VN_GetAt/F_VN_GetAt_SINT

	{attribute 'TcIecLibraryType'}
	{attribute 'external_name' := 'F_VN_GetAt_SINT_GUID_FFBBC736_76E0_2DF6_517D_6C42B79833FF'}
	(* Gets the SINT element at the specified index of the container. *)
	FUNCTION F_VN_GetAt_SINT : HRESULT
	VAR_INPUT
		ipContainer	:	ITcVnContainer;	(* Container with SINT elements *)
	END_VAR
	VAR_IN_OUT
		nElement	:	SINT;	(* Returns the element at the specified index *)
	END_VAR
	VAR_INPUT
		nIndex	:	ULINT;	(* Index of the requested element *)
		hrPrev	:	HRESULT;	(* HRESULT indicating the result of previous operations (If SUCCEEDED(hrPrev) equals false, no operation is executed.) *)
	END_VAR

END_FUNCTION

// Functions/Basic Container Operations/F_VN_GetAt/F_VN_GetAt_TcVnDMatch

	{attribute 'TcIecLibraryType'}
	{attribute 'external_name' := 'F_VN_GetAt_TcVnDMatch_GUID_45AA68A5_09F1_2884_77B2_F3B54B3F8A80'}
	(* Gets the TcVnDMatch element at the specified index of the container. *)
	FUNCTION F_VN_GetAt_TcVnDMatch : HRESULT
	VAR_INPUT
		ipContainer	:	ITcVnContainer;	(* Container with TcVnDMatch elements *)
	END_VAR
	VAR_IN_OUT
		stElement	:	TcVnDMatch;	(* Returns the element at the specified index *)
	END_VAR
	VAR_INPUT
		nIndex	:	ULINT;	(* Index of the requested element *)
		hrPrev	:	HRESULT;	(* HRESULT indicating the result of previous operations (If SUCCEEDED(hrPrev) equals false, no operation is executed.) *)
	END_VAR

END_FUNCTION

// Functions/Basic Container Operations/F_VN_GetAt/F_VN_GetAt_TcVnKeyPoint

	{attribute 'TcIecLibraryType'}
	{attribute 'external_name' := 'F_VN_GetAt_TcVnKeyPoint_GUID_5AA89398_758F_2C96_6BC2_5C301CAE1521'}
	(* Gets the TcVnKeyPoint element at the specified index of the container. *)
	FUNCTION F_VN_GetAt_TcVnKeyPoint : HRESULT
	VAR_INPUT
		ipContainer	:	ITcVnContainer;	(* Container with TcVnKeyPoint elements *)
	END_VAR
	VAR_IN_OUT
		stElement	:	TcVnKeyPoint;	(* Returns the element at the specified index *)
	END_VAR
	VAR_INPUT
		nIndex	:	ULINT;	(* Index of the requested element *)
		hrPrev	:	HRESULT;	(* HRESULT indicating the result of previous operations (If SUCCEEDED(hrPrev) equals false, no operation is executed.) *)
	END_VAR

END_FUNCTION

// Functions/Basic Container Operations/F_VN_GetAt/F_VN_GetAt_TcVnPoint2_DINT

	{attribute 'TcIecLibraryType'}
	{attribute 'external_name' := 'F_VN_GetAt_TcVnPoint2_DINT_GUID_9493A157_3E26_28BA_72A0_0392BA574485'}
	(* Gets the TcVnPoint2_DINT element at the specified index of the container. *)
	FUNCTION F_VN_GetAt_TcVnPoint2_DINT : HRESULT
	VAR_INPUT
		ipContainer	:	ITcVnContainer;	(* Container with TcVnPoint2_DINT elements *)
	END_VAR
	VAR_IN_OUT
		aElement	:	TcVnPoint2_DINT;	(* Returns the element at the specified index *)
	END_VAR
	VAR_INPUT
		nIndex	:	ULINT;	(* Index of the requested element *)
		hrPrev	:	HRESULT;	(* HRESULT indicating the result of previous operations (If SUCCEEDED(hrPrev) equals false, no operation is executed.) *)
	END_VAR

END_FUNCTION

// Functions/Basic Container Operations/F_VN_GetAt/F_VN_GetAt_TcVnPoint2_LREAL

	{attribute 'TcIecLibraryType'}
	{attribute 'external_name' := 'F_VN_GetAt_TcVnPoint2_LREAL_GUID_E946DE5F_3DD2_2DA1_50CD_5CFF3E171282'}
	(* Gets the TcVnPoint2_LREAL element at the specified index of the container. *)
	FUNCTION F_VN_GetAt_TcVnPoint2_LREAL : HRESULT
	VAR_INPUT
		ipContainer	:	ITcVnContainer;	(* Container with TcVnPoint2_LREAL elements *)
	END_VAR
	VAR_IN_OUT
		aElement	:	TcVnPoint2_LREAL;	(* Returns the element at the specified index *)
	END_VAR
	VAR_INPUT
		nIndex	:	ULINT;	(* Index of the requested element *)
		hrPrev	:	HRESULT;	(* HRESULT indicating the result of previous operations (If SUCCEEDED(hrPrev) equals false, no operation is executed.) *)
	END_VAR

END_FUNCTION

// Functions/Basic Container Operations/F_VN_GetAt/F_VN_GetAt_TcVnPoint2_REAL

	{attribute 'TcIecLibraryType'}
	{attribute 'external_name' := 'F_VN_GetAt_TcVnPoint2_REAL_GUID_40B32EDB_166B_2710_487E_F9022F94C2E6'}
	(* Gets the TcVnPoint2_REAL element at the specified index of the container. *)
	FUNCTION F_VN_GetAt_TcVnPoint2_REAL : HRESULT
	VAR_INPUT
		ipContainer	:	ITcVnContainer;	(* Container with TcVnPoint2_REAL elements *)
	END_VAR
	VAR_IN_OUT
		aElement	:	TcVnPoint2_REAL;	(* Returns the element at the specified index *)
	END_VAR
	VAR_INPUT
		nIndex	:	ULINT;	(* Index of the requested element *)
		hrPrev	:	HRESULT;	(* HRESULT indicating the result of previous operations (If SUCCEEDED(hrPrev) equals false, no operation is executed.) *)
	END_VAR

END_FUNCTION

// Functions/Basic Container Operations/F_VN_GetAt/F_VN_GetAt_TcVnPoint3_LREAL

	{attribute 'TcIecLibraryType'}
	{attribute 'external_name' := 'F_VN_GetAt_TcVnPoint3_LREAL_GUID_E7948DC1_4465_23BC_6638_CAA07618CD1C'}
	(* Gets the TcVnPoint3_LREAL element at the specified index of the container. *)
	FUNCTION F_VN_GetAt_TcVnPoint3_LREAL : HRESULT
	VAR_INPUT
		ipContainer	:	ITcVnContainer;	(* Container with TcVnPoint3_LREAL elements *)
	END_VAR
	VAR_IN_OUT
		aElement	:	TcVnPoint3_LREAL;	(* Returns the element at the specified index *)
	END_VAR
	VAR_INPUT
		nIndex	:	ULINT;	(* Index of the requested element *)
		hrPrev	:	HRESULT;	(* HRESULT indicating the result of previous operations (If SUCCEEDED(hrPrev) equals false, no operation is executed.) *)
	END_VAR

END_FUNCTION

// Functions/Basic Container Operations/F_VN_GetAt/F_VN_GetAt_TcVnPoint3_REAL

	{attribute 'TcIecLibraryType'}
	{attribute 'external_name' := 'F_VN_GetAt_TcVnPoint3_REAL_GUID_7DF04FAF_077C_2974_72A7_6585F1F80934'}
	(* Gets the TcVnPoint3_REAL element at the specified index of the container. *)
	FUNCTION F_VN_GetAt_TcVnPoint3_REAL : HRESULT
	VAR_INPUT
		ipContainer	:	ITcVnContainer;	(* Container with TcVnPoint3_REAL elements *)
	END_VAR
	VAR_IN_OUT
		aElement	:	TcVnPoint3_REAL;	(* Returns the element at the specified index *)
	END_VAR
	VAR_INPUT
		nIndex	:	ULINT;	(* Index of the requested element *)
		hrPrev	:	HRESULT;	(* HRESULT indicating the result of previous operations (If SUCCEEDED(hrPrev) equals false, no operation is executed.) *)
	END_VAR

END_FUNCTION

// Functions/Basic Container Operations/F_VN_GetAt/F_VN_GetAt_TcVnRectangle_DINT

	{attribute 'TcIecLibraryType'}
	{attribute 'external_name' := 'F_VN_GetAt_TcVnRectangle_DINT_GUID_021EC085_911E_2E72_74FE_E73B6AE55125'}
	(* Gets the TcVnRectangle_DINT element at the specified index of the container. *)
	FUNCTION F_VN_GetAt_TcVnRectangle_DINT : HRESULT
	VAR_INPUT
		ipContainer	:	ITcVnContainer;	(* Container with TcVnRectangle_DINT elements *)
	END_VAR
	VAR_IN_OUT
		stElement	:	TcVnRectangle_DINT;	(* Returns the element at the specified index *)
	END_VAR
	VAR_INPUT
		nIndex	:	ULINT;	(* Index of the requested element *)
		hrPrev	:	HRESULT;	(* HRESULT indicating the result of previous operations (If SUCCEEDED(hrPrev) equals false, no operation is executed.) *)
	END_VAR

END_FUNCTION

// Functions/Basic Container Operations/F_VN_GetAt/F_VN_GetAt_TcVnRotatedRectangle

	{attribute 'TcIecLibraryType'}
	{attribute 'external_name' := 'F_VN_GetAt_TcVnRotatedRectangle_GUID_4FBD28BF_E56A_2DDD_556D_846D702BBB66'}
	(* Gets the TcVnRotatedRectangle element at the specified index of the container. *)
	FUNCTION F_VN_GetAt_TcVnRotatedRectangle : HRESULT
	VAR_INPUT
		ipContainer	:	ITcVnContainer;	(* Container with TcVnRotatedRectangle elements *)
	END_VAR
	VAR_IN_OUT
		stElement	:	TcVnRotatedRectangle;	(* Returns the element at the specified index *)
	END_VAR
	VAR_INPUT
		nIndex	:	ULINT;	(* Index of the requested element *)
		hrPrev	:	HRESULT;	(* HRESULT indicating the result of previous operations (If SUCCEEDED(hrPrev) equals false, no operation is executed.) *)
	END_VAR

END_FUNCTION

// Functions/Basic Container Operations/F_VN_GetAt/F_VN_GetAt_TcVnVector2_DINT

	{attribute 'TcIecLibraryType'}
	{attribute 'external_name' := 'F_VN_GetAt_TcVnVector2_DINT_GUID_906F32BD_401A_2515_5CD6_D5FCB866480D'}
	(* Gets the TcVnVector2_DINT element at the specified index of the container. *)
	FUNCTION F_VN_GetAt_TcVnVector2_DINT : HRESULT
	VAR_INPUT
		ipContainer	:	ITcVnContainer;	(* Container with TcVnVector2_DINT elements *)
	END_VAR
	VAR_IN_OUT
		aElement	:	TcVnVector2_DINT;	(* Returns the element at the specified index *)
	END_VAR
	VAR_INPUT
		nIndex	:	ULINT;	(* Index of the requested element *)
		hrPrev	:	HRESULT;	(* HRESULT indicating the result of previous operations (If SUCCEEDED(hrPrev) equals false, no operation is executed.) *)
	END_VAR

END_FUNCTION

// Functions/Basic Container Operations/F_VN_GetAt/F_VN_GetAt_TcVnVector2_INT

	{attribute 'TcIecLibraryType'}
	{attribute 'external_name' := 'F_VN_GetAt_TcVnVector2_INT_GUID_07BCDE1A_2937_2697_685F_DDDB08A8CAE0'}
	(* Gets the TcVnVector2_INT element at the specified index of the container. *)
	FUNCTION F_VN_GetAt_TcVnVector2_INT : HRESULT
	VAR_INPUT
		ipContainer	:	ITcVnContainer;	(* Container with TcVnVector2_INT elements *)
	END_VAR
	VAR_IN_OUT
		aElement	:	TcVnVector2_INT;	(* Returns the element at the specified index *)
	END_VAR
	VAR_INPUT
		nIndex	:	ULINT;	(* Index of the requested element *)
		hrPrev	:	HRESULT;	(* HRESULT indicating the result of previous operations (If SUCCEEDED(hrPrev) equals false, no operation is executed.) *)
	END_VAR

END_FUNCTION

// Functions/Basic Container Operations/F_VN_GetAt/F_VN_GetAt_TcVnVector2_REAL

